LIN {X 0,Y 192.812,Z 326.454,A -85,B 0,C 180,E1 -21972.633,E2 -21972.633} C_VEL
LIN {X 0,Y 192.759,Z 326.462,A -85,B 0,C 180,E1 -21976.959,E2 -21976.959} C_VEL
LIN {X 0,Y 192.618,Z 326.481,A -85,B 0,C 180,E1 -21981.4,E2 -21981.4} C_VEL
LIN {X 0,Y 192.649,Z 326.477,A -85,B 0,C 180,E1 -21984.213,E2 -21984.213} C_VEL
LIN {X 0,Y 192.646,Z 326.478,A -85,B 0,C 180,E1 -21988.889,E2 -21988.889} C_VEL
LIN {X 0,Y 192.627,Z 326.525,A -85,B 0,C 180,E1 -21991.327,E2 -21991.327} C_VEL
LIN {X 0,Y 193.973,Z 330.689,A -85,B 0,C 180,E1 -21995.112,E2 -21995.112} C_VEL
LIN {X 0,Y 197.718,Z 336.194,A -85,B 0,C 180,E1 -21997.257,E2 -21997.257} C_VEL
LIN {X 0,Y 199.002,Z 337.882,A -85,B 0,C 180,E1 -21997.932,E2 -21997.932} C_VEL
LIN {X 0,Y 202.174,Z 342.489,A -85,B 0,C 180,E1 -21999.538,E2 -21999.538} C_VEL
LIN {X 0,Y 207.22,Z 350.444,A -85,B 0,C 180,E1 -22001.911,E2 -22001.911} C_VEL
LIN {X 0,Y 210.777,Z 356.31,A -85,B 0,C 180,E1 -22003.459,E2 -22003.459} C_VEL
LIN {X 0,Y 216.071,Z 365.771,A -85,B 0,C 180,E1 -22005.619,E2 -22005.619} C_VEL
LIN {X 0,Y 220.821,Z 375.163,A -85,B 0,C 180,E1 -22007.434,E2 -22007.434} C_VEL
LIN {X 0,Y 226.552,Z 388.01,A -85,B 0,C 180,E1 -22009.515,E2 -22009.515} C_VEL
LIN {X 0,Y 226.643,Z 388.254,A -85,B 0,C 180,E1 -22009.549,E2 -22009.549} C_VEL
LIN {X 0,Y 227.386,Z 391.769,A -85,B 0,C 180,E1 -22009.885,E2 -22009.885} C_VEL
LIN {X 0,Y 227.296,Z 396.569,A -85,B 0,C 180,E1 -22010.071,E2 -22010.071} C_VEL
LIN {X 0,Y 225.976,Z 403.4,A -85,B 0,C 180,E1 -22010.046,E2 -22010.046} C_VEL
LIN {X 0,Y 222.803,Z 415.633,A -85,B 0,C 180,E1 -22009.796,E2 -22009.796} C_VEL
LIN {X 0,Y 222.248,Z 419.787,A -85,B 0,C 180,E1 -22009.842,E2 -22009.842} C_VEL
LIN {X 0,Y 220.74,Z 442.418,A -85,B 0,C 180,E1 -22010.562,E2 -22010.562} C_VEL
LIN {X 0,Y 218.905,Z 456.037,A -85,B 0,C 180,E1 -22011.297,E2 -22011.297} C_VEL
LIN {X 0,Y 216.473,Z 467.79,A -85,B 0,C 180,E1 -22012.208,E2 -22012.208} C_VEL
LIN {X 0,Y 213.017,Z 480.41,A -85,B 0,C 180,E1 -22013.568,E2 -22013.568} C_VEL
LIN {X 0,Y 209.487,Z 491.624,A -85,B 0,C 180,E1 -22015.227,E2 -22015.227} C_VEL
LIN {X 0,Y 205.624,Z 501.768,A -85,B 0,C 180,E1 -22017.139,E2 -22017.139} C_VEL
LIN {X 0,Y 202.052,Z 510.095,A -85,B 0,C 180,E1 -22019.132,E2 -22019.132} C_VEL
LIN {X 0,Y 197.643,Z 519.156,A -85,B 0,C 180,E1 -22021.89,E2 -22021.89} C_VEL
LIN {X 0,Y 194.46,Z 525.362,A -85,B 0,C 180,E1 -22024.297,E2 -22024.297} C_VEL
LIN {X 0,Y 191.313,Z 531.467,A -85,B 0,C 180,E1 -22027.311,E2 -22027.311} C_VEL
LIN {X 0,Y 188.552,Z 536.333,A -85,B 0,C 180,E1 -22030.399,E2 -22030.399} C_VEL
LIN {X 0,Y 186.292,Z 540.098,A -85,B 0,C 180,E1 -22033.563,E2 -22033.563} C_VEL
LIN {X 0,Y 184.741,Z 542.869,A -85,B 0,C 180,E1 -22036.805,E2 -22036.805} C_VEL
LIN {X 0,Y 183.512,Z 545.134,A -85,B 0,C 180,E1 -22041.188,E2 -22041.188} C_VEL
LIN {X 0,Y 183.214,Z 545.672,A -85,B 0,C 180,E1 -22043.391,E2 -22043.391} C_VEL
LIN {X 0,Y 183.158,Z 545.528,A -85,B 0,C 180,E1 -22047.8,E2 -22047.8} C_VEL
LIN {X 0,Y 183.324,Z 544.879,A -85,B 0,C 180,E1 -22049.999,E2 -22049.999} C_VEL
LIN {X 0,Y 183.155,Z 542.674,A -85,B 0,C 180,E1 -22053.907,E2 -22053.907} C_VEL
LIN {X 0,Y 183.36,Z 539.178,A -85,B 0,C 180,E1 -22057.709,E2 -22057.709} C_VEL
LIN {X 0,Y 183.873,Z 534.991,A -85,B 0,C 180,E1 -22061.017,E2 -22061.017} C_VEL
LIN {X 0,Y 185.089,Z 528.586,A -85,B 0,C 180,E1 -22064.85,E2 -22064.85} C_VEL
LIN {X 0,Y 186.807,Z 521.607,A -85,B 0,C 180,E1 -22068.081,E2 -22068.081} C_VEL
LIN {X 0,Y 188.819,Z 513.433,A -85,B 0,C 180,E1 -22071.069,E2 -22071.069} C_VEL
LIN {X 0,Y 191.033,Z 503.806,A -85,B 0,C 180,E1 -22073.87,E2 -22073.87} C_VEL
LIN {X 0,Y 193.448,Z 493.911,A -85,B 0,C 180,E1 -22076.135,E2 -22076.135} C_VEL
LIN {X 0,Y 195.816,Z 482.985,A -85,B 0,C 180,E1 -22078.103,E2 -22078.103} C_VEL
LIN {X 0,Y 198.082,Z 470.698,A -85,B 0,C 180,E1 -22079.782,E2 -22079.782} C_VEL
LIN {X 0,Y 200.015,Z 457.808,A -85,B 0,C 180,E1 -22081.069,E2 -22081.069} C_VEL
LIN {X 0,Y 201.423,Z 444.674,A -85,B 0,C 180,E1 -22081.935,E2 -22081.935} C_VEL
LIN {X 0,Y 202.283,Z 426.501,A -85,B 0,C 180,E1 -22082.646,E2 -22082.646} C_VEL
LIN {X 0,Y 203.728,Z 391.931,A -85,B 0,C 180,E1 -22083.797,E2 -22083.797} C_VEL
LIN {X 0,Y 201.201,Z 366.378,A -85,B 0,C 180,E1 -22085.24,E2 -22085.24} C_VEL
LIN {X 0,Y 195.007,Z 350.312,A -85,B 0,C 180,E1 -22087.011,E2 -22087.011} C_VEL
LIN {X 0,Y 188.811,Z 336.625,A -85,B 0,C 180,E1 -22088.828,E2 -22088.828} C_VEL
LIN {X 0,Y 186.825,Z 332.463,A -85,B 0,C 180,E1 -22089.479,E2 -22089.479} C_VEL
LIN {X 0,Y 185.486,Z 327.381,A -85,B 0,C 180,E1 -22092.364,E2 -22092.364} C_VEL
LIN {X 0,Y 185.455,Z 327.384,A -85,B 0,C 180,E1 -22096.989,E2 -22096.989} C_VEL
LIN {X 0,Y 185.466,Z 327.383,A -85,B 0,C 180,E1 -22099.894,E2 -22099.894} C_VEL
LIN {X 0,Y 185.504,Z 327.38,A -85,B 0,C 180,E1 -22102.71,E2 -22102.71} C_VEL
LIN {X 0,Y 185.544,Z 327.374,A -85,B 0,C 180,E1 -22107.974,E2 -22107.974} C_VEL
LIN {X 0,Y 185.58,Z 327.371,A -85,B 0,C 180,E1 -22110.575,E2 -22110.575} C_VEL
LIN {X 0,Y 185.586,Z 327.368,A -85,B 0,C 180,E1 -22115.382,E2 -22115.382} C_VEL
LIN {X 0,Y 185.672,Z 327.356,A -85,B 0,C 180,E1 -22121.132,E2 -22121.132} C_VEL
LIN {X 0,Y 185.693,Z 327.354,A -85,B 0,C 180,E1 -22124.637,E2 -22124.637} C_VEL
LIN {X 0,Y 185.921,Z 327.301,A -85,B 0,C 180,E1 -22129.358,E2 -22129.358} C_VEL
LIN {X 0,Y 185.957,Z 327.322,A -85,B 0,C 180,E1 -22133.489,E2 -22133.489} C_VEL
LIN {X 0,Y 186.204,Z 327.27,A -85,B 0,C 180,E1 -22137.836,E2 -22137.836} C_VEL
LIN {X 0,Y 186.401,Z 327.242,A -85,B 0,C 180,E1 -22140,E2 -22140} C_VEL
LIN {X 0,Y 185.911,Z 327.327,A -85,B 0,C 180,E1 -22144.336,E2 -22144.336} C_VEL
LIN {X 0,Y 185.973,Z 327.298,A -85,B 0,C 180,E1 -22148.694,E2 -22148.694} C_VEL
LIN {X 0,Y 185.726,Z 327.345,A -85,B 0,C 180,E1 -22153.123,E2 -22153.123} C_VEL
LIN {X 0,Y 185.686,Z 327.347,A -85,B 0,C 180,E1 -22157.625,E2 -22157.625} C_VEL
LIN {X 0,Y 185.574,Z 327.354,A -85,B 0,C 180,E1 -22162.254,E2 -22162.254} C_VEL
LIN {X 0,Y 185.557,Z 327.366,A -85,B 0,C 180,E1 -22167.032,E2 -22167.032} C_VEL
LIN {X 0,Y 185.576,Z 327.347,A -85,B 0,C 180,E1 -22169.493,E2 -22169.493} C_VEL
LIN {X 0,Y 185.496,Z 327.379,A -85,B 0,C 180,E1 -22174.632,E2 -22174.632} C_VEL
LIN {X 0,Y 185.502,Z 327.365,A -85,B 0,C 180,E1 -22177.313,E2 -22177.313} C_VEL
LIN {X 0,Y 185.466,Z 327.372,A -85,B 0,C 180,E1 -22180.725,E2 -22180.725} C_VEL
LIN {X 0,Y 185.452,Z 327.368,A -85,B 0,C 180,E1 -22186.057,E2 -22186.057} C_VEL
LIN {X 0,Y 185.453,Z 327.382,A -85,B 0,C 180,E1 -22189.893,E2 -22189.893} C_VEL
LIN {X 0,Y 185.498,Z 327.371,A -85,B 0,C 180,E1 -22192.714,E2 -22192.714} C_VEL
LIN {X 0,Y 185.528,Z 327.373,A -85,B 0,C 180,E1 -22197.973,E2 -22197.973} C_VEL
LIN {X 0,Y 185.542,Z 327.365,A -85,B 0,C 180,E1 -22200.598,E2 -22200.598} C_VEL
LIN {X 0,Y 186.69,Z 330.413,A -85,B 0,C 180,E1 -22201.032,E2 -22201.032} C_VEL
LIN {X 0,Y 188.069,Z 332.496,A -85,B 0,C 180,E1 -22201.42,E2 -22201.42} C_VEL
LIN {X 0,Y 196.411,Z 347.504,A -85,B 0,C 180,E1 -22203.72,E2 -22203.72} C_VEL
LIN {X 0,Y 202.022,Z 359.493,A -85,B 0,C 180,E1 -22205.209,E2 -22205.209} C_VEL
LIN {X 0,Y 204.649,Z 366.895,A -85,B 0,C 180,E1 -22205.944,E2 -22205.944} C_VEL
LIN {X 0,Y 202.081,Z 428.474,A -85,B 0,C 180,E1 -22208.047,E2 -22208.047} C_VEL
LIN {X 0,Y 201.051,Z 441.583,A -85,B 0,C 180,E1 -22208.871,E2 -22208.871} C_VEL
LIN {X 0,Y 199.598,Z 454.209,A -85,B 0,C 180,E1 -22210.057,E2 -22210.057} C_VEL
LIN {X 0,Y 197.638,Z 466.289,A -85,B 0,C 180,E1 -22211.604,E2 -22211.604} C_VEL
LIN {X 0,Y 195.28,Z 476.551,A -85,B 0,C 180,E1 -22213.268,E2 -22213.268} C_VEL
LIN {X 0,Y 193.014,Z 487.091,A -85,B 0,C 180,E1 -22215.504,E2 -22215.504} C_VEL
LIN {X 0,Y 190.864,Z 495.73,A -85,B 0,C 180,E1 -22217.777,E2 -22217.777} C_VEL
LIN {X 0,Y 188.847,Z 503.679,A -85,B 0,C 180,E1 -22220.36,E2 -22220.36} C_VEL
LIN {X 0,Y 186.807,Z 511.476,A -85,B 0,C 180,E1 -22223.52,E2 -22223.52} C_VEL
LIN {X 0,Y 185.331,Z 517.701,A -85,B 0,C 180,E1 -22226.74,E2 -22226.74} C_VEL
LIN {X 0,Y 184.203,Z 522.666,A -85,B 0,C 180,E1 -22230.001,E2 -22230.001} C_VEL
LIN {X 0,Y 183.672,Z 526.498,A -85,B 0,C 180,E1 -22233.291,E2 -22233.291} C_VEL
LIN {X 0,Y 183.237,Z 529.33,A -85,B 0,C 180,E1 -22236.608,E2 -22236.608} C_VEL
LIN {X 0,Y 183.023,Z 531.63,A -85,B 0,C 180,E1 -22241.07,E2 -22241.07} C_VEL
LIN {X 0,Y 183.204,Z 532.178,A -85,B 0,C 180,E1 -22243.308,E2 -22243.308} C_VEL
LIN {X 0,Y 183.963,Z 532.117,A -85,B 0,C 180,E1 -22247.239,E2 -22247.239} C_VEL
LIN {X 0,Y 184.736,Z 531.333,A -85,B 0,C 180,E1 -22250.023,E2 -22250.023} C_VEL
LIN {X 0,Y 185.631,Z 530.231,A -85,B 0,C 180,E1 -22252.248,E2 -22252.248} C_VEL
LIN {X 0,Y 187.811,Z 527.22,A -85,B 0,C 180,E1 -22256.092,E2 -22256.092} C_VEL
LIN {X 0,Y 190.685,Z 522.809,A -85,B 0,C 180,E1 -22259.84,E2 -22259.84} C_VEL
LIN {X 0,Y 193.663,Z 517.741,A -85,B 0,C 180,E1 -22262.981,E2 -22262.981} C_VEL
LIN {X 0,Y 197.251,Z 511.31,A -85,B 0,C 180,E1 -22266.008,E2 -22266.008} C_VEL
LIN {X 0,Y 201.297,Z 503.198,A -85,B 0,C 180,E1 -22268.936,E2 -22268.936} C_VEL
LIN {X 0,Y 205.47,Z 494.072,A -85,B 0,C 180,E1 -22271.474,E2 -22271.474} C_VEL
LIN {X 0,Y 209.165,Z 484.669,A -85,B 0,C 180,E1 -22273.536,E2 -22273.536} C_VEL
LIN {X 0,Y 212.535,Z 474.439,A -85,B 0,C 180,E1 -22275.313,E2 -22275.313} C_VEL
LIN {X 0,Y 215.81,Z 462.836,A -85,B 0,C 180,E1 -22276.853,E2 -22276.853} C_VEL
LIN {X 0,Y 218.392,Z 450.783,A -85,B 0,C 180,E1 -22278.084,E2 -22278.084} C_VEL
LIN {X 0,Y 220.382,Z 437.633,A -85,B 0,C 180,E1 -22279.034,E2 -22279.034} C_VEL
LIN {X 0,Y 221.649,Z 425.884,A -85,B 0,C 180,E1 -22279.552,E2 -22279.552} C_VEL
LIN {X 0,Y 224.092,Z 386.328,A -85,B 0,C 180,E1 -22280.719,E2 -22280.719} C_VEL
LIN {X 0,Y 218.281,Z 374.069,A -85,B 0,C 180,E1 -22282.866,E2 -22282.866} C_VEL
LIN {X 0,Y 213.163,Z 365.33,A -85,B 0,C 180,E1 -22284.835,E2 -22284.835} C_VEL
LIN {X 0,Y 206.43,Z 355.119,A -85,B 0,C 180,E1 -22287.646,E2 -22287.646} C_VEL
LIN {X 0,Y 203.304,Z 350.827,A -85,B 0,C 180,E1 -22289.056,E2 -22289.056} C_VEL
LIN {X 0,Y 200.397,Z 346.848,A -85,B 0,C 180,E1 -22290.451,E2 -22290.451} C_VEL
LIN {X 0,Y 197.599,Z 343.03,A -85,B 0,C 180,E1 -22291.884,E2 -22291.884} C_VEL
LIN {X 0,Y 194.884,Z 339.672,A -85,B 0,C 180,E1 -22293.351,E2 -22293.351} C_VEL
LIN {X 0,Y 194.108,Z 338.344,A -85,B 0,C 180,E1 -22293.816,E2 -22293.816} C_VEL
LIN {X 0,Y 191.552,Z 336.002,A -85,B 0,C 180,E1 -22295.269,E2 -22295.269} C_VEL
LIN {X 0,Y 189.931,Z 332.999,A -85,B 0,C 180,E1 -22296.363,E2 -22296.363} C_VEL
LIN {X 0,Y 187.274,Z 331.168,A -85,B 0,C 180,E1 -22298.031,E2 -22298.031} C_VEL
LIN {X 0,Y 185.951,Z 328.94,A -85,B 0,C 180,E1 -22299.031,E2 -22299.031} C_VEL
LIN {X 0,Y 185.571,Z 327.359,A -85,B 0,C 180,E1 -22299.494,E2 -22299.494} C_VEL
LIN {X 0,Y 185.691,Z 327.352,A -85,B 0,C 180,E1 -22302.376,E2 -22302.376} C_VEL
LIN {X 0,Y 185.767,Z 327.346,A -85,B 0,C 180,E1 -22306.88,E2 -22306.88} C_VEL
LIN {X 0,Y 186.031,Z 327.313,A -85,B 0,C 180,E1 -22311.309,E2 -22311.309} C_VEL
LIN {X 0,Y 186.209,Z 327.275,A -85,B 0,C 180,E1 -22317.837,E2 -22317.837} C_VEL
LIN {X 0,Y 186.406,Z 327.262,A -85,B 0,C 180,E1 -22320,E2 -22320} C_VEL
LIN {X 0,Y 185.926,Z 327.319,A -85,B 0,C 180,E1 -22324.336,E2 -22324.336} C_VEL
LIN {X 0,Y 186.011,Z 327.306,A -85,B 0,C 180,E1 -22328.693,E2 -22328.693} C_VEL
LIN {X 0,Y 185.736,Z 327.34,A -85,B 0,C 180,E1 -22333.123,E2 -22333.123} C_VEL
LIN {X 0,Y 185.692,Z 327.347,A -85,B 0,C 180,E1 -22337.625,E2 -22337.625} C_VEL
LIN {X 0,Y 185.58,Z 327.366,A -85,B 0,C 180,E1 -22342.254,E2 -22342.254} C_VEL
LIN {X 0,Y 185.561,Z 327.369,A -85,B 0,C 180,E1 -22347.033,E2 -22347.033} C_VEL
LIN {X 0,Y 185.635,Z 327.541,A -85,B 0,C 180,E1 -22348.245,E2 -22348.245} C_VEL
LIN {X 0,Y 186.616,Z 330.253,A -85,B 0,C 180,E1 -22351.029,E2 -22351.029} C_VEL
LIN {X 0,Y 189.543,Z 334.692,A -85,B 0,C 180,E1 -22353.09,E2 -22353.09} C_VEL
LIN {X 0,Y 191.645,Z 337.156,A -85,B 0,C 180,E1 -22354.401,E2 -22354.401} C_VEL
LIN {X 0,Y 195.551,Z 342.71,A -85,B 0,C 180,E1 -22356.706,E2 -22356.706} C_VEL
LIN {X 0,Y 200.091,Z 349.688,A -85,B 0,C 180,E1 -22359.135,E2 -22359.135} C_VEL
LIN {X 0,Y 204.237,Z 356.412,A -85,B 0,C 180,E1 -22361.159,E2 -22361.159} C_VEL
LIN {X 0,Y 208.864,Z 364.216,A -85,B 0,C 180,E1 -22363.239,E2 -22363.239} C_VEL
LIN {X 0,Y 214.944,Z 375.86,A -85,B 0,C 180,E1 -22365.78,E2 -22365.78} C_VEL
LIN {X 0,Y 221.35,Z 390.268,A -85,B 0,C 180,E1 -22368.276,E2 -22368.276} C_VEL
LIN {X 0,Y 222.965,Z 394.781,A -85,B 0,C 180,E1 -22368.906,E2 -22368.906} C_VEL
LIN {X 0,Y 223.453,Z 400.102,A -85,B 0,C 180,E1 -22369.269,E2 -22369.269} C_VEL
LIN {X 0,Y 222.248,Z 419.787,A -85,B 0,C 180,E1 -22369.842,E2 -22369.842} C_VEL
LIN {X 0,Y 221.384,Z 425.64,A -85,B 0,C 180,E1 -22369.875,E2 -22369.875} C_VEL
LIN {X 0,Y 215.811,Z 444.62,A -85,B 0,C 180,E1 -22369.47,E2 -22369.47} C_VEL
LIN {X 0,Y 214.644,Z 450.37,A -85,B 0,C 180,E1 -22369.66,E2 -22369.66} C_VEL
LIN {X 0,Y 212.192,Z 463.375,A -85,B 0,C 180,E1 -22370.55,E2 -22370.55} C_VEL
LIN {X 0,Y 208.901,Z 476.223,A -85,B 0,C 180,E1 -22371.816,E2 -22371.816} C_VEL
LIN {X 0,Y 205.574,Z 486.943,A -85,B 0,C 180,E1 -22373.253,E2 -22373.253} C_VEL
LIN {X 0,Y 201.41,Z 497.92,A -85,B 0,C 180,E1 -22375.152,E2 -22375.152} C_VEL
LIN {X 0,Y 196.79,Z 508.622,A -85,B 0,C 180,E1 -22377.608,E2 -22377.608} C_VEL
LIN {X 0,Y 192.878,Z 516.543,A -85,B 0,C 180,E1 -22379.932,E2 -22379.932} C_VEL
LIN {X 0,Y 188.701,Z 524.322,A -85,B 0,C 180,E1 -22382.855,E2 -22382.855} C_VEL
LIN {X 0,Y 184.775,Z 531.477,A -85,B 0,C 180,E1 -22386.46,E2 -22386.46} C_VEL
LIN {X 0,Y 181.842,Z 536.282,A -85,B 0,C 180,E1 -22389.644,E2 -22389.644} C_VEL
LIN {X 0,Y 179.473,Z 539.992,A -85,B 0,C 180,E1 -22392.92,E2 -22392.92} C_VEL
LIN {X 0,Y 177.801,Z 542.712,A -85,B 0,C 180,E1 -22396.28,E2 -22396.28} C_VEL
LIN {X 0,Y 176.474,Z 544.927,A -85,B 0,C 180,E1 -22400.833,E2 -22400.833} C_VEL
LIN {X 0,Y 176.142,Z 545.418,A -85,B 0,C 180,E1 -22403.125,E2 -22403.125} C_VEL
LIN {X 0,Y 176.054,Z 545.227,A -85,B 0,C 180,E1 -22407.711,E2 -22407.711} C_VEL
LIN {X 0,Y 176.243,Z 544.555,A -85,B 0,C 180,E1 -22409.999,E2 -22409.999} C_VEL
LIN {X 0,Y 176.07,Z 542.538,A -85,B 0,C 180,E1 -22413.704,E2 -22413.704} C_VEL
LIN {X 0,Y 176.316,Z 538.726,A -85,B 0,C 180,E1 -22418.019,E2 -22418.019} C_VEL
LIN {X 0,Y 176.881,Z 534.483,A -85,B 0,C 180,E1 -22421.458,E2 -22421.458} C_VEL
LIN {X 0,Y 178.182,Z 528.015,A -85,B 0,C 180,E1 -22425.44,E2 -22425.44} C_VEL
LIN {X 0,Y 179.981,Z 520.946,A -85,B 0,C 180,E1 -22428.792,E2 -22428.792} C_VEL
LIN {X 0,Y 181.807,Z 514.255,A -85,B 0,C 180,E1 -22431.344,E2 -22431.344} C_VEL
LIN {X 0,Y 184.017,Z 504.925,A -85,B 0,C 180,E1 -22434.239,E2 -22434.239} C_VEL
LIN {X 0,Y 186.763,Z 494.121,A -85,B 0,C 180,E1 -22436.843,E2 -22436.843} C_VEL
LIN {X 0,Y 189.215,Z 483.345,A -85,B 0,C 180,E1 -22438.871,E2 -22438.871} C_VEL
LIN {X 0,Y 191.571,Z 471.237,A -85,B 0,C 180,E1 -22440.597,E2 -22440.597} C_VEL
LIN {X 0,Y 193.57,Z 458.603,A -85,B 0,C 180,E1 -22441.918,E2 -22441.918} C_VEL
LIN {X 0,Y 195.02,Z 446.072,A -85,B 0,C 180,E1 -22442.818,E2 -22442.818} C_VEL
LIN {X 0,Y 195.868,Z 430.553,A -85,B 0,C 180,E1 -22443.486,E2 -22443.486} C_VEL
LIN {X 0,Y 197.525,Z 391.561,A -85,B 0,C 180,E1 -22444.825,E2 -22444.825} C_VEL
LIN {X 0,Y 195.125,Z 368.319,A -85,B 0,C 180,E1 -22446.22,E2 -22446.22} C_VEL
LIN {X 0,Y 189.403,Z 353.427,A -85,B 0,C 180,E1 -22447.953,E2 -22447.953} C_VEL
LIN {X 0,Y 183.653,Z 340.606,A -85,B 0,C 180,E1 -22449.74,E2 -22449.74} C_VEL
LIN {X 0,Y 180.545,Z 334.628,A -85,B 0,C 180,E1 -22450.724,E2 -22450.724} C_VEL
LIN {X 0,Y 179.412,Z 332.121,A -85,B 0,C 180,E1 -22451.162,E2 -22451.162} C_VEL
LIN {X 0,Y 178.406,Z 328.263,A -85,B 0,C 180,E1 -22453.563,E2 -22453.563} C_VEL
LIN {X 0,Y 178.401,Z 328.267,A -85,B 0,C 180,E1 -22458.458,E2 -22458.458} C_VEL
LIN {X 0,Y 178.421,Z 328.264,A -85,B 0,C 180,E1 -22463.782,E2 -22463.782} C_VEL
LIN {X 0,Y 178.485,Z 328.256,A -85,B 0,C 180,E1 -22466.546,E2 -22466.546} C_VEL
LIN {X 0,Y 178.521,Z 328.25,A -85,B 0,C 180,E1 -22470.005,E2 -22470.005} C_VEL
LIN {X 0,Y 178.533,Z 328.246,A -85,B 0,C 180,E1 -22474.875,E2 -22474.875} C_VEL
LIN {X 0,Y 178.621,Z 328.236,A -85,B 0,C 180,E1 -22480.783,E2 -22480.783} C_VEL
LIN {X 0,Y 178.658,Z 328.221,A -85,B 0,C 180,E1 -22486.347,E2 -22486.347} C_VEL
LIN {X 0,Y 178.956,Z 328.181,A -85,B 0,C 180,E1 -22490.962,E2 -22490.962} C_VEL
LIN {X 0,Y 179.15,Z 328.148,A -85,B 0,C 180,E1 -22497.751,E2 -22497.751} C_VEL
LIN {X 0,Y 179.364,Z 328.117,A -85,B 0,C 180,E1 -22500,E2 -22500} C_VEL
LIN {X 0,Y 178.858,Z 328.205,A -85,B 0,C 180,E1 -22504.507,E2 -22504.507} C_VEL
LIN {X 0,Y 178.903,Z 328.175,A -85,B 0,C 180,E1 -22509.04,E2 -22509.04} C_VEL
LIN {X 0,Y 178.654,Z 328.227,A -85,B 0,C 180,E1 -22513.652,E2 -22513.652} C_VEL
LIN {X 0,Y 178.617,Z 328.214,A -85,B 0,C 180,E1 -22519.214,E2 -22519.214} C_VEL
LIN {X 0,Y 178.516,Z 328.248,A -85,B 0,C 180,E1 -22525.114,E2 -22525.114} C_VEL
LIN {X 0,Y 178.52,Z 328.223,A -85,B 0,C 180,E1 -22529.994,E2 -22529.994} C_VEL
LIN {X 0,Y 178.482,Z 328.25,A -85,B 0,C 180,E1 -22534.22,E2 -22534.22} C_VEL
LIN {X 0,Y 178.391,Z 328.243,A -85,B 0,C 180,E1 -22539.075,E2 -22539.075} C_VEL
LIN {X 0,Y 178.394,Z 328.26,A -85,B 0,C 180,E1 -22542.046,E2 -22542.046} C_VEL
LIN {X 0,Y 178.388,Z 328.249,A -85,B 0,C 180,E1 -22545.165,E2 -22545.165} C_VEL
LIN {X 0,Y 178.394,Z 328.261,A -85,B 0,C 180,E1 -22548.462,E2 -22548.462} C_VEL
LIN {X 0,Y 178.416,Z 328.261,A -85,B 0,C 180,E1 -22553.783,E2 -22553.783} C_VEL
LIN {X 0,Y 178.463,Z 328.253,A -85,B 0,C 180,E1 -22558.549,E2 -22558.549} C_VEL
LIN {X 0,Y 178.486,Z 328.413,A -85,B 0,C 180,E1 -22559.078,E2 -22559.078} C_VEL
LIN {X 0,Y 179.518,Z 331.187,A -85,B 0,C 180,E1 -22559.46,E2 -22559.46} C_VEL
LIN {X 0,Y 181.038,Z 333.344,A -85,B 0,C 180,E1 -22559.918,E2 -22559.918} C_VEL
LIN {X 0,Y 188.944,Z 347.167,A -85,B 0,C 180,E1 -22562.265,E2 -22562.265} C_VEL
LIN {X 0,Y 195.661,Z 360.844,A -85,B 0,C 180,E1 -22564.151,E2 -22564.151} C_VEL
LIN {X 0,Y 198.582,Z 369.012,A -85,B 0,C 180,E1 -22565.012,E2 -22565.012} C_VEL
LIN {X 0,Y 195.826,Z 429.016,A -85,B 0,C 180,E1 -22567.098,E2 -22567.098} C_VEL
LIN {X 0,Y 194.675,Z 442.788,A -85,B 0,C 180,E1 -22568.005,E2 -22568.005} C_VEL
LIN {X 0,Y 193.13,Z 455.173,A -85,B 0,C 180,E1 -22569.22,E2 -22569.22} C_VEL
LIN {X 0,Y 191.258,Z 466.259,A -85,B 0,C 180,E1 -22570.689,E2 -22570.689} C_VEL
LIN {X 0,Y 188.816,Z 476.575,A -85,B 0,C 180,E1 -22572.398,E2 -22572.398} C_VEL
LIN {X 0,Y 186.426,Z 487.157,A -85,B 0,C 180,E1 -22574.7,E2 -22574.7} C_VEL
LIN {X 0,Y 183.967,Z 496.715,A -85,B 0,C 180,E1 -22577.312,E2 -22577.312} C_VEL
LIN {X 0,Y 181.858,Z 504.545,A -85,B 0,C 180,E1 -22579.986,E2 -22579.986} C_VEL
LIN {X 0,Y 179.764,Z 512.194,A -85,B 0,C 180,E1 -22583.265,E2 -22583.265} C_VEL
LIN {X 0,Y 178.248,Z 518.333,A -85,B 0,C 180,E1 -22586.61,E2 -22586.61} C_VEL
LIN {X 0,Y 177.095,Z 523.22,A -85,B 0,C 180,E1 -22590.001,E2 -22590.001} C_VEL
LIN {X 0,Y 176.57,Z 526.98,A -85,B 0,C 180,E1 -22593.424,E2 -22593.424} C_VEL
LIN {X 0,Y 176.105,Z 529.746,A -85,B 0,C 180,E1 -22596.877,E2 -22596.877} C_VEL
LIN {X 0,Y 175.923,Z 531.061,A -85,B 0,C 180,E1 -22599.196,E2 -22599.196} C_VEL
LIN {X 0,Y 175.941,Z 531.981,A -85,B 0,C 180,E1 -22601.522,E2 -22601.522} C_VEL
LIN {X 0,Y 176.172,Z 532.465,A -85,B 0,C 180,E1 -22603.849,E2 -22603.849} C_VEL
LIN {X 0,Y 176.929,Z 532.409,A -85,B 0,C 180,E1 -22607.575,E2 -22607.575} C_VEL
LIN {X 0,Y 177.9,Z 531.517,A -85,B 0,C 180,E1 -22610.828,E2 -22610.828} C_VEL
LIN {X 0,Y 178.894,Z 530.351,A -85,B 0,C 180,E1 -22613.133,E2 -22613.133} C_VEL
LIN {X 0,Y 181.06,Z 527.583,A -85,B 0,C 180,E1 -22616.778,E2 -22616.778} C_VEL
LIN {X 0,Y 184.368,Z 522.785,A -85,B 0,C 180,E1 -22620.972,E2 -22620.972} C_VEL
LIN {X 0,Y 188.19,Z 516.555,A -85,B 0,C 180,E1 -22624.756,E2 -22624.756} C_VEL
LIN {X 0,Y 192.051,Z 509.823,A -85,B 0,C 180,E1 -22627.804,E2 -22627.804} C_VEL
LIN {X 0,Y 196.386,Z 501.542,A -85,B 0,C 180,E1 -22630.687,E2 -22630.687} C_VEL
LIN {X 0,Y 200.529,Z 492.509,A -85,B 0,C 180,E1 -22633.112,E2 -22633.112} C_VEL
LIN {X 0,Y 204.369,Z 482.778,A -85,B 0,C 180,E1 -22635.176,E2 -22635.176} C_VEL
LIN {X 0,Y 207.96,Z 472.084,A -85,B 0,C 180,E1 -22636.955,E2 -22636.955} C_VEL
LIN {X 0,Y 211.264,Z 460.038,A -85,B 0,C 180,E1 -22638.481,E2 -22638.481} C_VEL
LIN {X 0,Y 213.751,Z 448.236,A -85,B 0,C 180,E1 -22639.592,E2 -22639.592} C_VEL
LIN {X 0,Y 215.627,Z 435.138,A -85,B 0,C 180,E1 -22640.486,E2 -22640.486} C_VEL
LIN {X 0,Y 216.929,Z 422.502,A -85,B 0,C 180,E1 -22640.954,E2 -22640.954} C_VEL
LIN {X 0,Y 219.055,Z 388.94,A -85,B 0,C 180,E1 -22641.943,E2 -22641.943} C_VEL
LIN {X 0,Y 213.27,Z 376.764,A -85,B 0,C 180,E1 -22644.221,E2 -22644.221} C_VEL
LIN {X 0,Y 206.554,Z 365.622,A -85,B 0,C 180,E1 -22647.017,E2 -22647.017} C_VEL
LIN {X 0,Y 200.616,Z 356.921,A -85,B 0,C 180,E1 -22649.745,E2 -22649.745} C_VEL
LIN {X 0,Y 197.256,Z 352.324,A -85,B 0,C 180,E1 -22651.432,E2 -22651.432} C_VEL
LIN {X 0,Y 194.692,Z 348.815,A -85,B 0,C 180,E1 -22652.815,E2 -22652.815} C_VEL
LIN {X 0,Y 191.985,Z 345.144,A -85,B 0,C 180,E1 -22654.379,E2 -22654.379} C_VEL
LIN {X 0,Y 188.631,Z 341.293,A -85,B 0,C 180,E1 -22656.436,E2 -22656.436} C_VEL
LIN {X 0,Y 187.551,Z 339.461,A -85,B 0,C 180,E1 -22657.191,E2 -22657.191} C_VEL
LIN {X 0,Y 184.902,Z 337.157,A -85,B 0,C 180,E1 -22658.979,E2 -22658.979} C_VEL
LIN {X 0,Y 183.244,Z 334.042,A -85,B 0,C 180,E1 -22660.342,E2 -22660.342} C_VEL
LIN {X 0,Y 180.561,Z 332.251,A -85,B 0,C 180,E1 -22662.443,E2 -22662.443} C_VEL
LIN {X 0,Y 179.044,Z 329.903,A -85,B 0,C 180,E1 -22663.906,E2 -22663.906} C_VEL
LIN {X 0,Y 178.648,Z 328.22,A -85,B 0,C 180,E1 -22664.455,E2 -22664.455} C_VEL
LIN {X 0,Y 178.897,Z 328.188,A -85,B 0,C 180,E1 -22669.154,E2 -22669.154} C_VEL
LIN {X 0,Y 178.935,Z 328.183,A -85,B 0,C 180,E1 -22673.234,E2 -22673.234} C_VEL
LIN {X 0,Y 179.155,Z 328.154,A -85,B 0,C 180,E1 -22677.752,E2 -22677.752} C_VEL
LIN {X 0,Y 179.37,Z 328.139,A -85,B 0,C 180,E1 -22680,E2 -22680} C_VEL
LIN {X 0,Y 178.875,Z 328.199,A -85,B 0,C 180,E1 -22684.507,E2 -22684.507} C_VEL
LIN {X 0,Y 178.962,Z 328.187,A -85,B 0,C 180,E1 -22689.038,E2 -22689.038} C_VEL
LIN {X 0,Y 178.663,Z 328.226,A -85,B 0,C 180,E1 -22693.652,E2 -22693.652} C_VEL
LIN {X 0,Y 178.623,Z 328.226,A -85,B 0,C 180,E1 -22699.214,E2 -22699.214} C_VEL
LIN {X 0,Y 178.547,Z 328.389,A -85,B 0,C 180,E1 -22704.218,E2 -22704.218} C_VEL
LIN {X 0,Y 178.79,Z 329.503,A -85,B 0,C 180,E1 -22705.374,E2 -22705.374} C_VEL
LIN {X 0,Y 179.919,Z 331.705,A -85,B 0,C 180,E1 -22706.537,E2 -22706.537} C_VEL
LIN {X 0,Y 182.072,Z 333.998,A -85,B 0,C 180,E1 -22708.377,E2 -22708.377} C_VEL
LIN {X 0,Y 184.724,Z 337.012,A -85,B 0,C 180,E1 -22710.431,E2 -22710.431} C_VEL
LIN {X 0,Y 187.504,Z 341.164,A -85,B 0,C 180,E1 -22712.455,E2 -22712.455} C_VEL
LIN {X 0,Y 189.341,Z 343.472,A -85,B 0,C 180,E1 -22713.657,E2 -22713.657} C_VEL
LIN {X 0,Y 193.636,Z 349.968,A -85,B 0,C 180,E1 -22716.304,E2 -22716.304} C_VEL
LIN {X 0,Y 197.297,Z 355.702,A -85,B 0,C 180,E1 -22718.339,E2 -22718.339} C_VEL
LIN {X 0,Y 200.988,Z 361.812,A -85,B 0,C 180,E1 -22720.233,E2 -22720.233} C_VEL
LIN {X 0,Y 205.088,Z 368.897,A -85,B 0,C 180,E1 -22722.181,E2 -22722.181} C_VEL
LIN {X 0,Y 211.007,Z 380.548,A -85,B 0,C 180,E1 -22724.802,E2 -22724.802} C_VEL
LIN {X 0,Y 216.816,Z 393.894,A -85,B 0,C 180,E1 -22727.202,E2 -22727.202} C_VEL
LIN {X 0,Y 218.117,Z 397.454,A -85,B 0,C 180,E1 -22727.734,E2 -22727.734} C_VEL
LIN {X 0,Y 218.387,Z 401.64,A -85,B 0,C 180,E1 -22728.004,E2 -22728.004} C_VEL
LIN {X 0,Y 215.767,Z 441.266,A -85,B 0,C 180,E1 -22729.217,E2 -22729.217} C_VEL
LIN {X 0,Y 214.644,Z 450.37,A -85,B 0,C 180,E1 -22729.66,E2 -22729.66} C_VEL
LIN {X 0,Y 213.27,Z 456.065,A -85,B 0,C 180,E1 -22729.876,E2 -22729.876} C_VEL
LIN {X 0,Y 209.323,Z 465.152,A -85,B 0,C 180,E1 -22730.035,E2 -22730.035} C_VEL
LIN {X 0,Y 204.86,Z 473.938,A -85,B 0,C 180,E1 -22730.359,E2 -22730.359} C_VEL
LIN {X 0,Y 202.69,Z 479.163,A -85,B 0,C 180,E1 -22730.844,E2 -22730.844} C_VEL
LIN {X 0,Y 198.523,Z 491.391,A -85,B 0,C 180,E1 -22732.681,E2 -22732.681} C_VEL
LIN {X 0,Y 194.292,Z 501.467,A -85,B 0,C 180,E1 -22734.636,E2 -22734.636} C_VEL
LIN {X 0,Y 190.009,Z 510.567,A -85,B 0,C 180,E1 -22736.936,E2 -22736.936} C_VEL
LIN {X 0,Y 185.253,Z 519.458,A -85,B 0,C 180,E1 -22739.823,E2 -22739.823} C_VEL
LIN {X 0,Y 181.06,Z 526.74,A -85,B 0,C 180,E1 -22742.927,E2 -22742.927} C_VEL
LIN {X 0,Y 177.177,Z 533.196,A -85,B 0,C 180,E1 -22746.629,E2 -22746.629} C_VEL
LIN {X 0,Y 174.304,Z 537.567,A -85,B 0,C 180,E1 -22749.956,E2 -22749.956} C_VEL
LIN {X 0,Y 171.955,Z 540.887,A -85,B 0,C 180,E1 -22753.375,E2 -22753.375} C_VEL
LIN {X 0,Y 170.057,Z 543.833,A -85,B 0,C 180,E1 -22758.074,E2 -22758.074} C_VEL
LIN {X 0,Y 169.456,Z 544.712,A -85,B 0,C 180,E1 -22760.45,E2 -22760.45} C_VEL
LIN {X 0,Y 168.932,Z 545.236,A -85,B 0,C 180,E1 -22765.226,E2 -22765.226} C_VEL
LIN {X 0,Y 168.952,Z 544.925,A -85,B 0,C 180,E1 -22767.615,E2 -22767.615} C_VEL
LIN {X 0,Y 169.144,Z 544.228,A -85,B 0,C 180,E1 -22769.999,E2 -22769.999} C_VEL
LIN {X 0,Y 168.976,Z 542.428,A -85,B 0,C 180,E1 -22773.427,E2 -22773.427} C_VEL
LIN {X 0,Y 169.15,Z 539.47,A -85,B 0,C 180,E1 -22777.159,E2 -22777.159} C_VEL
LIN {X 0,Y 169.63,Z 535.544,A -85,B 0,C 180,E1 -22780.744,E2 -22780.744} C_VEL
LIN {X 0,Y 170.559,Z 530.459,A -85,B 0,C 180,E1 -22784.313,E2 -22784.313} C_VEL
LIN {X 0,Y 172.259,Z 524.069,A -85,B 0,C 180,E1 -22787.817,E2 -22787.817} C_VEL
LIN {X 0,Y 174.075,Z 517.531,A -85,B 0,C 180,E1 -22790.686,E2 -22790.686} C_VEL
LIN {X 0,Y 176.124,Z 509.635,A -85,B 0,C 180,E1 -22793.517,E2 -22793.517} C_VEL
LIN {X 0,Y 178.676,Z 499.984,A -85,B 0,C 180,E1 -22796.263,E2 -22796.263} C_VEL
LIN {X 0,Y 181.346,Z 489.273,A -85,B 0,C 180,E1 -22798.657,E2 -22798.657} C_VEL
LIN {X 0,Y 183.701,Z 478.932,A -85,B 0,C 180,E1 -22800.457,E2 -22800.457} C_VEL
LIN {X 0,Y 185.881,Z 467.736,A -85,B 0,C 180,E1 -22801.959,E2 -22801.959} C_VEL
LIN {X 0,Y 187.748,Z 455.138,A -85,B 0,C 180,E1 -22803.192,E2 -22803.192} C_VEL
LIN {X 0,Y 189.097,Z 442.028,A -85,B 0,C 180,E1 -22804.05,E2 -22804.05} C_VEL
LIN {X 0,Y 191.417,Z 392.633,A -85,B 0,C 180,E1 -22805.848,E2 -22805.848} C_VEL
LIN {X 0,Y 189.205,Z 370.499,A -85,B 0,C 180,E1 -22807.232,E2 -22807.232} C_VEL
LIN {X 0,Y 183.098,Z 354.582,A -85,B 0,C 180,E1 -22809.206,E2 -22809.206} C_VEL
LIN {X 0,Y 178.04,Z 343.54,A -85,B 0,C 180,E1 -22810.874,E2 -22810.874} C_VEL
LIN {X 0,Y 173.759,Z 335.362,A -85,B 0,C 180,E1 -22812.332,E2 -22812.332} C_VEL
LIN {X 0,Y 172.051,Z 331.735,A -85,B 0,C 180,E1 -22813.043,E2 -22813.043} C_VEL
LIN {X 0,Y 171.375,Z 329.137,A -85,B 0,C 180,E1 -22814.814,E2 -22814.814} C_VEL
LIN {X 0,Y 171.333,Z 329.145,A -85,B 0,C 180,E1 -22818.98,E2 -22818.98} C_VEL
LIN {X 0,Y 171.385,Z 329.139,A -85,B 0,C 180,E1 -22822.04,E2 -22822.04} C_VEL
LIN {X 0,Y 171.397,Z 329.137,A -85,B 0,C 180,E1 -22825.091,E2 -22825.091} C_VEL
LIN {X 0,Y 171.447,Z 329.132,A -85,B 0,C 180,E1 -22830.533,E2 -22830.533} C_VEL
LIN {X 0,Y 171.456,Z 329.129,A -85,B 0,C 180,E1 -22835.801,E2 -22835.801} C_VEL
LIN {X 0,Y 171.577,Z 329.113,A -85,B 0,C 180,E1 -22840.871,E2 -22840.871} C_VEL
LIN {X 0,Y 171.576,Z 329.106,A -85,B 0,C 180,E1 -22845.772,E2 -22845.772} C_VEL
LIN {X 0,Y 171.885,Z 329.056,A -85,B 0,C 180,E1 -22850.586,E2 -22850.586} C_VEL
LIN {X 0,Y 171.817,Z 329.08,A -85,B 0,C 180,E1 -22855.307,E2 -22855.307} C_VEL
LIN {X 0,Y 172.327,Z 328.992,A -85,B 0,C 180,E1 -22859.999,E2 -22859.999} C_VEL
LIN {X 0,Y 171.806,Z 329.083,A -85,B 0,C 180,E1 -22864.692,E2 -22864.692} C_VEL
LIN {X 0,Y 171.841,Z 329.052,A -85,B 0,C 180,E1 -22869.415,E2 -22869.415} C_VEL
LIN {X 0,Y 171.572,Z 329.112,A -85,B 0,C 180,E1 -22874.227,E2 -22874.227} C_VEL
LIN {X 0,Y 171.536,Z 329.092,A -85,B 0,C 180,E1 -22879.557,E2 -22879.557} C_VEL
LIN {X 0,Y 171.455,Z 329.127,A -85,B 0,C 180,E1 -22885.609,E2 -22885.609} C_VEL
LIN {X 0,Y 171.438,Z 329.105,A -85,B 0,C 180,E1 -22890.587,E2 -22890.587} C_VEL
LIN {X 0,Y 171.389,Z 329.134,A -85,B 0,C 180,E1 -22895.035,E2 -22895.035} C_VEL
LIN {X 0,Y 171.353,Z 329.118,A -85,B 0,C 180,E1 -22898.807,E2 -22898.807} C_VEL
LIN {X 0,Y 171.316,Z 329.136,A -85,B 0,C 180,E1 -22904.218,E2 -22904.218} C_VEL
LIN {X 0,Y 171.327,Z 329.144,A -85,B 0,C 180,E1 -22908.98,E2 -22908.98} C_VEL
LIN {X 0,Y 171.357,Z 329.129,A -85,B 0,C 180,E1 -22912.035,E2 -22912.035} C_VEL
LIN {X 0,Y 171.444,Z 329.127,A -85,B 0,C 180,E1 -22917.298,E2 -22917.298} C_VEL
LIN {X 0,Y 172.418,Z 331.942,A -85,B 0,C 180,E1 -22917.739,E2 -22917.739} C_VEL
LIN {X 0,Y 174.115,Z 334.367,A -85,B 0,C 180,E1 -22918.3,E2 -22918.3} C_VEL
LIN {X 0,Y 181.199,Z 346.338,A -85,B 0,C 180,E1 -22920.578,E2 -22920.578} C_VEL
LIN {X 0,Y 187.777,Z 359.058,A -85,B 0,C 180,E1 -22922.566,E2 -22922.566} C_VEL
LIN {X 0,Y 191.684,Z 368.126,A -85,B 0,C 180,E1 -22923.729,E2 -22923.729} C_VEL
LIN {X 0,Y 192.342,Z 369.991,A -85,B 0,C 180,E1 -22923.934,E2 -22923.934} C_VEL
LIN {X 0,Y 189.625,Z 429.501,A -85,B 0,C 180,E1 -22926.087,E2 -22926.087} C_VEL
LIN {X 0,Y 188.43,Z 443.194,A -85,B 0,C 180,E1 -22927.018,E2 -22927.018} C_VEL
LIN {X 0,Y 186.725,Z 456.05,A -85,B 0,C 180,E1 -22928.327,E2 -22928.327} C_VEL
LIN {X 0,Y 184.482,Z 467.811,A -85,B 0,C 180,E1 -22929.95,E2 -22929.95} C_VEL
LIN {X 0,Y 181.803,Z 479.152,A -85,B 0,C 180,E1 -22931.986,E2 -22931.986} C_VEL
LIN {X 0,Y 179.318,Z 489.331,A -85,B 0,C 180,E1 -22934.369,E2 -22934.369} C_VEL
LIN {X 0,Y 176.578,Z 499.301,A -85,B 0,C 180,E1 -22937.356,E2 -22937.356} C_VEL
LIN {X 0,Y 174.115,Z 508.075,A -85,B 0,C 180,E1 -22940.709,E2 -22940.709} C_VEL
LIN {X 0,Y 172.155,Z 515.096,A -85,B 0,C 180,E1 -22944.143,E2 -22944.143} C_VEL
LIN {X 0,Y 170.777,Z 520.7,A -85,B 0,C 180,E1 -22947.642,E2 -22947.642} C_VEL
LIN {X 0,Y 169.782,Z 525.124,A -85,B 0,C 180,E1 -22951.187,E2 -22951.187} C_VEL
LIN {X 0,Y 169.316,Z 528.657,A -85,B 0,C 180,E1 -22955.004,E2 -22955.004} C_VEL
LIN {X 0,Y 168.813,Z 531.444,A -85,B 0,C 180,E1 -22959.587,E2 -22959.587} C_VEL
LIN {X 0,Y 168.869,Z 532.318,A -85,B 0,C 180,E1 -22962.011,E2 -22962.011} C_VEL
LIN {X 0,Y 169.167,Z 532.75,A -85,B 0,C 180,E1 -22964.435,E2 -22964.435} C_VEL
LIN {X 0,Y 169.922,Z 532.697,A -85,B 0,C 180,E1 -22967.959,E2 -22967.959} C_VEL
LIN {X 0,Y 171.107,Z 531.684,A -85,B 0,C 180,E1 -22971.696,E2 -22971.696} C_VEL
LIN {X 0,Y 172.212,Z 530.472,A -85,B 0,C 180,E1 -22974.086,E2 -22974.086} C_VEL
LIN {X 0,Y 174.353,Z 527.938,A -85,B 0,C 180,E1 -22977.527,E2 -22977.527} C_VEL
LIN {X 0,Y 177.12,Z 524.201,A -85,B 0,C 180,E1 -22981.054,E2 -22981.054} C_VEL
LIN {X 0,Y 180.359,Z 519.37,A -85,B 0,C 180,E1 -22984.404,E2 -22984.404} C_VEL
LIN {X 0,Y 184.23,Z 513.223,A -85,B 0,C 180,E1 -22987.617,E2 -22987.617} C_VEL
LIN {X 0,Y 188.625,Z 505.528,A -85,B 0,C 180,E1 -22990.696,E2 -22990.696} C_VEL
LIN {X 0,Y 192.831,Z 497.351,A -85,B 0,C 180,E1 -22993.204,E2 -22993.204} C_VEL
LIN {X 0,Y 197.084,Z 487.838,A -85,B 0,C 180,E1 -22995.496,E2 -22995.496} C_VEL
LIN {X 0,Y 201.136,Z 476.928,A -85,B 0,C 180,E1 -22997.574,E2 -22997.574} C_VEL
LIN {X 0,Y 204.524,Z 466.295,A -85,B 0,C 180,E1 -22999.111,E2 -22999.111} C_VEL
LIN {X 0,Y 207.698,Z 453.366,A -85,B 0,C 180,E1 -23000.527,E2 -23000.527} C_VEL
LIN {X 0,Y 209.999,Z 440.536,A -85,B 0,C 180,E1 -23001.537,E2 -23001.537} C_VEL
LIN {X 0,Y 211.474,Z 428.246,A -85,B 0,C 180,E1 -23002.158,E2 -23002.158} C_VEL
LIN {X 0,Y 214.006,Z 391.247,A -85,B 0,C 180,E1 -23003.276,E2 -23003.276} C_VEL
LIN {X 0,Y 209.023,Z 380.827,A -85,B 0,C 180,E1 -23005.359,E2 -23005.359} C_VEL
LIN {X 0,Y 202.899,Z 370.544,A -85,B 0,C 180,E1 -23008.06,E2 -23008.06} C_VEL
LIN {X 0,Y 197.574,Z 362.538,A -85,B 0,C 180,E1 -23010.645,E2 -23010.645} C_VEL
LIN {X 0,Y 192.383,Z 355.162,A -85,B 0,C 180,E1 -23013.471,E2 -23013.471} C_VEL
LIN {X 0,Y 188.821,Z 350.522,A -85,B 0,C 180,E1 -23015.621,E2 -23015.621} C_VEL
LIN {X 0,Y 186.104,Z 347.132,A -85,B 0,C 180,E1 -23017.409,E2 -23017.409} C_VEL
LIN {X 0,Y 185.099,Z 345.71,A -85,B 0,C 180,E1 -23018.126,E2 -23018.126} C_VEL
LIN {X 0,Y 182.428,Z 342.89,A -85,B 0,C 180,E1 -23020.081,E2 -23020.081} C_VEL
LIN {X 0,Y 181.125,Z 340.599,A -85,B 0,C 180,E1 -23021.201,E2 -23021.201} C_VEL
LIN {X 0,Y 178.364,Z 338.271,A -85,B 0,C 180,E1 -23023.549,E2 -23023.549} C_VEL
LIN {X 0,Y 176.907,Z 335.547,A -85,B 0,C 180,E1 -23025.109,E2 -23025.109} C_VEL
LIN {X 0,Y 176.743,Z 335.054,A -85,B 0,C 180,E1 -23025.316,E2 -23025.316} C_VEL
LIN {X 0,Y 174.049,Z 333.472,A -85,B 0,C 180,E1 -23028.205,E2 -23028.205} C_VEL
LIN {X 0,Y 172.403,Z 330.952,A -85,B 0,C 180,E1 -23030.546,E2 -23030.546} C_VEL
LIN {X 0,Y 171.896,Z 329.071,A -85,B 0,C 180,E1 -23031.625,E2 -23031.625} C_VEL
LIN {X 0,Y 172.103,Z 329.032,A -85,B 0,C 180,E1 -23037.66,E2 -23037.66} C_VEL
LIN {X 0,Y 172.333,Z 329.015,A -85,B 0,C 180,E1 -23040.001,E2 -23040.001} C_VEL
LIN {X 0,Y 171.824,Z 329.078,A -85,B 0,C 180,E1 -23044.693,E2 -23044.693} C_VEL
LIN {X 0,Y 171.89,Z 329.071,A -85,B 0,C 180,E1 -23049.413,E2 -23049.413} C_VEL
LIN {X 0,Y 171.58,Z 329.108,A -85,B 0,C 180,E1 -23054.227,E2 -23054.227} C_VEL
LIN {X 0,Y 171.59,Z 329.28,A -85,B 0,C 180,E1 -23057.582,E2 -23057.582} C_VEL
LIN {X 0,Y 172.628,Z 332.072,A -85,B 0,C 180,E1 -23059.458,E2 -23059.458} C_VEL
LIN {X 0,Y 174.777,Z 334.304,A -85,B 0,C 180,E1 -23062.222,E2 -23062.222} C_VEL
LIN {X 0,Y 176.747,Z 335.479,A -85,B 0,C 180,E1 -23064.276,E2 -23064.276} C_VEL
LIN {X 0,Y 178.215,Z 338.27,A -85,B 0,C 180,E1 -23065.866,E2 -23065.866} C_VEL
LIN {X 0,Y 180.761,Z 341.14,A -85,B 0,C 180,E1 -23068.127,E2 -23068.127} C_VEL
LIN {X 0,Y 182.624,Z 343.384,A -85,B 0,C 180,E1 -23069.633,E2 -23069.633} C_VEL
LIN {X 0,Y 185.571,Z 347.721,A -85,B 0,C 180,E1 -23071.861,E2 -23071.861} C_VEL
LIN {X 0,Y 187.384,Z 350.287,A -85,B 0,C 180,E1 -23073.111,E2 -23073.111} C_VEL
LIN {X 0,Y 190.961,Z 355.858,A -85,B 0,C 180,E1 -23075.417,E2 -23075.417} C_VEL
LIN {X 0,Y 194.538,Z 361.651,A -85,B 0,C 180,E1 -23077.513,E2 -23077.513} C_VEL
LIN {X 0,Y 199.394,Z 369.878,A -85,B 0,C 180,E1 -23080.089,E2 -23080.089} C_VEL
LIN {X 0,Y 205.287,Z 381.288,A -85,B 0,C 180,E1 -23082.941,E2 -23082.941} C_VEL
LIN {X 0,Y 210.276,Z 392.494,A -85,B 0,C 180,E1 -23085.186,E2 -23085.186} C_VEL
LIN {X 0,Y 213.39,Z 400.176,A -85,B 0,C 180,E1 -23086.519,E2 -23086.519} C_VEL
LIN {X 0,Y 213.419,Z 403.24,A -85,B 0,C 180,E1 -23086.678,E2 -23086.678} C_VEL
LIN {X 0,Y 210.76,Z 441.566,A -85,B 0,C 180,E1 -23087.875,E2 -23087.875} C_VEL
LIN {X 0,Y 208.852,Z 454.872,A -85,B 0,C 180,E1 -23088.589,E2 -23088.589} C_VEL
LIN {X 0,Y 206.009,Z 467.733,A -85,B 0,C 180,E1 -23089.595,E2 -23089.595} C_VEL
LIN {X 0,Y 202.69,Z 479.163,A -85,B 0,C 180,E1 -23090.844,E2 -23090.844} C_VEL
LIN {X 0,Y 200.418,Z 484.359,A -85,B 0,C 180,E1 -23091.403,E2 -23091.403} C_VEL
LIN {X 0,Y 195.253,Z 492.442,A -85,B 0,C 180,E1 -23092.155,E2 -23092.155} C_VEL
LIN {X 0,Y 189.888,Z 500.039,A -85,B 0,C 180,E1 -23093.122,E2 -23093.122} C_VEL
LIN {X 0,Y 187.339,Z 504.412,A -85,B 0,C 180,E1 -23094.016,E2 -23094.016} C_VEL
LIN {X 0,Y 183.283,Z 512.425,A -85,B 0,C 180,E1 -23096.22,E2 -23096.22} C_VEL
LIN {X 0,Y 178.385,Z 520.889,A -85,B 0,C 180,E1 -23099.191,E2 -23099.191} C_VEL
LIN {X 0,Y 174.174,Z 527.705,A -85,B 0,C 180,E1 -23102.353,E2 -23102.353} C_VEL
LIN {X 0,Y 170.676,Z 533.179,A -85,B 0,C 180,E1 -23105.683,E2 -23105.683} C_VEL
LIN {X 0,Y 167.635,Z 537.492,A -85,B 0,C 180,E1 -23109.123,E2 -23109.123} C_VEL
LIN {X 0,Y 165.146,Z 540.759,A -85,B 0,C 180,E1 -23112.668,E2 -23112.668} C_VEL
LIN {X 0,Y 163.098,Z 543.654,A -85,B 0,C 180,E1 -23117.557,E2 -23117.557} C_VEL
LIN {X 0,Y 162.433,Z 544.486,A -85,B 0,C 180,E1 -23120.033,E2 -23120.033} C_VEL
LIN {X 0,Y 161.851,Z 544.959,A -85,B 0,C 180,E1 -23125.017,E2 -23125.017} C_VEL
LIN {X 0,Y 161.867,Z 544.624,A -85,B 0,C 180,E1 -23127.511,E2 -23127.511} C_VEL
LIN {X 0,Y 162.046,Z 543.889,A -85,B 0,C 180,E1 -23129.999,E2 -23129.999} C_VEL
LIN {X 0,Y 161.883,Z 542.329,A -85,B 0,C 180,E1 -23133.103,E2 -23133.103} C_VEL
LIN {X 0,Y 162.069,Z 539.039,A -85,B 0,C 180,E1 -23137.474,E2 -23137.474} C_VEL
LIN {X 0,Y 162.606,Z 535.057,A -85,B 0,C 180,E1 -23141.214,E2 -23141.214} C_VEL
LIN {X 0,Y 163.922,Z 528.908,A -85,B 0,C 180,E1 -23145.542,E2 -23145.542} C_VEL
LIN {X 0,Y 165.803,Z 522.177,A -85,B 0,C 180,E1 -23149.177,E2 -23149.177} C_VEL
LIN {X 0,Y 168.149,Z 514.055,A -85,B 0,C 180,E1 -23152.635,E2 -23152.635} C_VEL
LIN {X 0,Y 170.533,Z 505.165,A -85,B 0,C 180,E1 -23155.639,E2 -23155.639} C_VEL
LIN {X 0,Y 173.493,Z 494.514,A -85,B 0,C 180,E1 -23158.422,E2 -23158.422} C_VEL
LIN {X 0,Y 176.136,Z 483.944,A -85,B 0,C 180,E1 -23160.579,E2 -23160.579} C_VEL
LIN {X 0,Y 178.675,Z 472.262,A -85,B 0,C 180,E1 -23162.405,E2 -23162.405} C_VEL
LIN {X 0,Y 180.82,Z 460.102,A -85,B 0,C 180,E1 -23163.798,E2 -23163.798} C_VEL
LIN {X 0,Y 182.53,Z 446.859,A -85,B 0,C 180,E1 -23164.856,E2 -23164.856} C_VEL
LIN {X 0,Y 183.442,Z 433.95,A -85,B 0,C 180,E1 -23165.494,E2 -23165.494} C_VEL
LIN {X 0,Y 185.371,Z 393.296,A -85,B 0,C 180,E1 -23166.957,E2 -23166.957} C_VEL
LIN {X 0,Y 183.415,Z 372.878,A -85,B 0,C 180,E1 -23168.286,E2 -23168.286} C_VEL
LIN {X 0,Y 177.323,Z 356.938,A -85,B 0,C 180,E1 -23170.384,E2 -23170.384} C_VEL
LIN {X 0,Y 171.774,Z 344.774,A -85,B 0,C 180,E1 -23172.352,E2 -23172.352} C_VEL
LIN {X 0,Y 166.702,Z 335.454,A -85,B 0,C 180,E1 -23174.216,E2 -23174.216} C_VEL
LIN {X 0,Y 164.668,Z 331.553,A -85,B 0,C 180,E1 -23175.019,E2 -23175.019} C_VEL
LIN {X 0,Y 164.277,Z 330.025,A -85,B 0,C 180,E1 -23176.191,E2 -23176.191} C_VEL
LIN {X 0,Y 164.294,Z 330.022,A -85,B 0,C 180,E1 -23180.351,E2 -23180.351} C_VEL
LIN {X 0,Y 164.328,Z 330.019,A -85,B 0,C 180,E1 -23186.221,E2 -23186.221} C_VEL
LIN {X 0,Y 164.404,Z 330.009,A -85,B 0,C 180,E1 -23189.137,E2 -23189.137} C_VEL
LIN {X 0,Y 164.415,Z 330.004,A -85,B 0,C 180,E1 -23194.693,E2 -23194.693} C_VEL
LIN {X 0,Y 164.482,Z 329.996,A -85,B 0,C 180,E1 -23200.05,E2 -23200.05} C_VEL
LIN {X 0,Y 164.523,Z 329.988,A -85,B 0,C 180,E1 -23205.149,E2 -23205.149} C_VEL
LIN {X 0,Y 164.799,Z 329.934,A -85,B 0,C 180,E1 -23210.178,E2 -23210.178} C_VEL
LIN {X 0,Y 164.847,Z 329.948,A -85,B 0,C 180,E1 -23212.651,E2 -23212.651} C_VEL
LIN {X 0,Y 165.046,Z 329.905,A -85,B 0,C 180,E1 -23217.559,E2 -23217.559} C_VEL
LIN {X 0,Y 165.29,Z 329.868,A -85,B 0,C 180,E1 -23219.999,E2 -23219.999} C_VEL
LIN {X 0,Y 164.755,Z 329.962,A -85,B 0,C 180,E1 -23224.894,E2 -23224.894} C_VEL
LIN {X 0,Y 164.822,Z 329.94,A -85,B 0,C 180,E1 -23227.349,E2 -23227.349} C_VEL
LIN {X 0,Y 164.699,Z 329.944,A -85,B 0,C 180,E1 -23231.059,E2 -23231.059} C_VEL
LIN {X 0,Y 164.479,Z 329.988,A -85,B 0,C 180,E1 -23237.403,E2 -23237.403} C_VEL
LIN {X 0,Y 164.469,Z 329.97,A -85,B 0,C 180,E1 -23239.989,E2 -23239.989} C_VEL
LIN {X 0,Y 164.382,Z 330.008,A -85,B 0,C 180,E1 -23246.128,E2 -23246.128} C_VEL
LIN {X 0,Y 164.372,Z 329.987,A -85,B 0,C 180,E1 -23251.228,E2 -23251.228} C_VEL
LIN {X 0,Y 164.291,Z 330.008,A -85,B 0,C 180,E1 -23256.79,E2 -23256.79} C_VEL
LIN {X 0,Y 164.287,Z 330.002,A -85,B 0,C 180,E1 -23259.917,E2 -23259.917} C_VEL
LIN {X 0,Y 164.276,Z 330.018,A -85,B 0,C 180,E1 -23263.342,E2 -23263.342} C_VEL
LIN {X 0,Y 164.257,Z 330.009,A -85,B 0,C 180,E1 -23266.799,E2 -23266.799} C_VEL
LIN {X 0,Y 164.286,Z 330.015,A -85,B 0,C 180,E1 -23270.355,E2 -23270.355} C_VEL
LIN {X 0,Y 164.369,Z 330.009,A -85,B 0,C 180,E1 -23275.373,E2 -23275.373} C_VEL
LIN {X 0,Y 165.366,Z 332.854,A -85,B 0,C 180,E1 -23275.847,E2 -23275.847} C_VEL
LIN {X 0,Y 167.157,Z 335.126,A -85,B 0,C 180,E1 -23276.485,E2 -23276.485} C_VEL
LIN {X 0,Y 175.193,Z 348.599,A -85,B 0,C 180,E1 -23279.29,E2 -23279.29} C_VEL
LIN {X 0,Y 181.994,Z 361.61,A -85,B 0,C 180,E1 -23281.478,E2 -23281.478} C_VEL
LIN {X 0,Y 186.13,Z 371.292,A -85,B 0,C 180,E1 -23282.789,E2 -23282.789} C_VEL
LIN {X 0,Y 186.303,Z 373.719,A -85,B 0,C 180,E1 -23282.934,E2 -23282.934} C_VEL
LIN {X 0,Y 183.523,Z 429.452,A -85,B 0,C 180,E1 -23284.976,E2 -23284.976} C_VEL
LIN {X 0,Y 182.32,Z 442.85,A -85,B 0,C 180,E1 -23285.899,E2 -23285.899} C_VEL
LIN {X 0,Y 180.544,Z 455.901,A -85,B 0,C 180,E1 -23287.243,E2 -23287.243} C_VEL
LIN {X 0,Y 178.206,Z 467.755,A -85,B 0,C 180,E1 -23288.909,E2 -23288.909} C_VEL
LIN {X 0,Y 175.403,Z 479.157,A -85,B 0,C 180,E1 -23291.002,E2 -23291.002} C_VEL
LIN {X 0,Y 172.798,Z 489.388,A -85,B 0,C 180,E1 -23293.46,E2 -23293.46} C_VEL
LIN {X 0,Y 170.164,Z 498.588,A -85,B 0,C 180,E1 -23296.263,E2 -23296.263} C_VEL
LIN {X 0,Y 167.522,Z 507.525,A -85,B 0,C 180,E1 -23299.73,E2 -23299.73} C_VEL
LIN {X 0,Y 165.39,Z 514.73,A -85,B 0,C 180,E1 -23303.29,E2 -23303.29} C_VEL
LIN {X 0,Y 164.095,Z 519.586,A -85,B 0,C 180,E1 -23306.318,E2 -23306.318} C_VEL
LIN {X 0,Y 162.894,Z 524.32,A -85,B 0,C 180,E1 -23310.001,E2 -23310.001} C_VEL
LIN {X 0,Y 162.508,Z 526.866,A -85,B 0,C 180,E1 -23312.48,E2 -23312.48} C_VEL
LIN {X 0,Y 162.215,Z 528.92,A -85,B 0,C 180,E1 -23314.972,E2 -23314.972} C_VEL
LIN {X 0,Y 161.852,Z 530.575,A -85,B 0,C 180,E1 -23317.486,E2 -23317.486} C_VEL
LIN {X 0,Y 161.726,Z 531.825,A -85,B 0,C 180,E1 -23320.011,E2 -23320.011} C_VEL
LIN {X 0,Y 161.81,Z 532.637,A -85,B 0,C 180,E1 -23322.544,E2 -23322.544} C_VEL
LIN {X 0,Y 162.184,Z 533.034,A -85,B 0,C 180,E1 -23325.071,E2 -23325.071} C_VEL
LIN {X 0,Y 162.9,Z 532.989,A -85,B 0,C 180,E1 -23328.353,E2 -23328.353} C_VEL
LIN {X 0,Y 164.351,Z 531.839,A -85,B 0,C 180,E1 -23332.636,E2 -23332.636} C_VEL
LIN {X 0,Y 165.593,Z 530.594,A -85,B 0,C 180,E1 -23335.114,E2 -23335.114} C_VEL
LIN {X 0,Y 167.642,Z 528.316,A -85,B 0,C 180,E1 -23338.313,E2 -23338.313} C_VEL
LIN {X 0,Y 170.886,Z 524.179,A -85,B 0,C 180,E1 -23342.321,E2 -23342.321} C_VEL
LIN {X 0,Y 174.357,Z 519.308,A -85,B 0,C 180,E1 -23345.736,E2 -23345.736} C_VEL
LIN {X 0,Y 178.504,Z 513.035,A -85,B 0,C 180,E1 -23349.047,E2 -23349.047} C_VEL
LIN {X 0,Y 183.158,Z 505.203,A -85,B 0,C 180,E1 -23352.183,E2 -23352.183} C_VEL
LIN {X 0,Y 187.743,Z 496.572,A -85,B 0,C 180,E1 -23354.814,E2 -23354.814} C_VEL
LIN {X 0,Y 192.49,Z 486.144,A -85,B 0,C 180,E1 -23357.29,E2 -23357.29} C_VEL
LIN {X 0,Y 196.29,Z 476.138,A -85,B 0,C 180,E1 -23359.14,E2 -23359.14} C_VEL
LIN {X 0,Y 200.26,Z 463.688,A -85,B 0,C 180,E1 -23360.862,E2 -23360.862} C_VEL
LIN {X 0,Y 203.069,Z 452.157,A -85,B 0,C 180,E1 -23362.08,E2 -23362.08} C_VEL
LIN {X 0,Y 205.341,Z 439.236,A -85,B 0,C 180,E1 -23363.062,E2 -23363.062} C_VEL
LIN {X 0,Y 206.829,Z 426.874,A -85,B 0,C 180,E1 -23363.634,E2 -23363.634} C_VEL
LIN {X 0,Y 209.13,Z 393.823,A -85,B 0,C 180,E1 -23364.645,E2 -23364.645} C_VEL
LIN {X 0,Y 204.952,Z 385.036,A -85,B 0,C 180,E1 -23366.505,E2 -23366.505} C_VEL
LIN {X 0,Y 199.003,Z 375.019,A -85,B 0,C 180,E1 -23369.29,E2 -23369.29} C_VEL
LIN {X 0,Y 194.448,Z 367.991,A -85,B 0,C 180,E1 -23371.645,E2 -23371.645} C_VEL
LIN {X 0,Y 189.547,Z 360.892,A -85,B 0,C 180,E1 -23374.467,E2 -23374.467} C_VEL
LIN {X 0,Y 186.325,Z 356.576,A -85,B 0,C 180,E1 -23376.522,E2 -23376.522} C_VEL
LIN {X 0,Y 183.499,Z 352.684,A -85,B 0,C 180,E1 -23378.516,E2 -23378.516} C_VEL
LIN {X 0,Y 180.24,Z 348.944,A -85,B 0,C 180,E1 -23381.028,E2 -23381.028} C_VEL
LIN {X 0,Y 179.149,Z 347.124,A -85,B 0,C 180,E1 -23382.005,E2 -23382.005} C_VEL
LIN {X 0,Y 176.439,Z 344.502,A -85,B 0,C 180,E1 -23384.478,E2 -23384.478} C_VEL
LIN {X 0,Y 175.053,Z 341.855,A -85,B 0,C 180,E1 -23386.062,E2 -23386.062} C_VEL
LIN {X 0,Y 172.474,Z 339.993,A -85,B 0,C 180,E1 -23389.034,E2 -23389.034} C_VEL
LIN {X 0,Y 170.853,Z 337.158,A -85,B 0,C 180,E1 -23391.574,E2 -23391.574} C_VEL
LIN {X 0,Y 170.497,Z 336.028,A -85,B 0,C 180,E1 -23392.302,E2 -23392.302} C_VEL
LIN {X 0,Y 167.903,Z 334.768,A -85,B 0,C 180,E1 -23397.602,E2 -23397.602} C_VEL
LIN {X 0,Y 167.254,Z 333.944,A -85,B 0,C 180,E1 -23400.001,E2 -23400.001} C_VEL
LIN {X 0,Y 166.888,Z 334.119,A -85,B 0,C 180,E1 -23407.867,E2 -23407.867} C_VEL
LIN {X 0,Y 170.279,Z 336.263,A -85,B 0,C 180,E1 -23416.948,E2 -23416.948} C_VEL
LIN {X 0,Y 171.66,Z 339.396,A -85,B 0,C 180,E1 -23419.421,E2 -23419.421} C_VEL
LIN {X 0,Y 174.085,Z 341.517,A -85,B 0,C 180,E1 -23422.475,E2 -23422.475} C_VEL
LIN {X 0,Y 175.073,Z 342.171,A -85,B 0,C 180,E1 -23423.535,E2 -23423.535} C_VEL
LIN {X 0,Y 176.874,Z 345.256,A -85,B 0,C 180,E1 -23425.52,E2 -23425.52} C_VEL
LIN {X 0,Y 180.251,Z 349.092,A -85,B 0,C 180,E1 -23428.531,E2 -23428.531} C_VEL
LIN {X 0,Y 183.141,Z 353.688,A -85,B 0,C 180,E1 -23430.882,E2 -23430.882} C_VEL
LIN {X 0,Y 184.886,Z 356.174,A -85,B 0,C 180,E1 -23432.153,E2 -23432.153} C_VEL
LIN {X 0,Y 188.431,Z 361.906,A -85,B 0,C 180,E1 -23434.568,E2 -23434.568} C_VEL
LIN {X 0,Y 191.813,Z 367.569,A -85,B 0,C 180,E1 -23436.657,E2 -23436.657} C_VEL
LIN {X 0,Y 196.697,Z 376.284,A -85,B 0,C 180,E1 -23439.389,E2 -23439.389} C_VEL
LIN {X 0,Y 202.067,Z 387.019,A -85,B 0,C 180,E1 -23442.115,E2 -23442.115} C_VEL
LIN {X 0,Y 207.627,Z 400.209,A -85,B 0,C 180,E1 -23444.743,E2 -23444.743} C_VEL
LIN {X 0,Y 208.687,Z 403.35,A -85,B 0,C 180,E1 -23445.244,E2 -23445.244} C_VEL
LIN {X 0,Y 205.943,Z 441.318,A -85,B 0,C 180,E1 -23446.441,E2 -23446.441} C_VEL
LIN {X 0,Y 203.908,Z 454.986,A -85,B 0,C 180,E1 -23447.184,E2 -23447.184} C_VEL
LIN {X 0,Y 200.953,Z 467.716,A -85,B 0,C 180,E1 -23448.188,E2 -23448.188} C_VEL
LIN {X 0,Y 197.426,Z 479.403,A -85,B 0,C 180,E1 -23449.487,E2 -23449.487} C_VEL
LIN {X 0,Y 193.418,Z 490.641,A -85,B 0,C 180,E1 -23451.185,E2 -23451.185} C_VEL
LIN {X 0,Y 189.027,Z 500.823,A -85,B 0,C 180,E1 -23453.163,E2 -23453.163} C_VEL
LIN {X 0,Y 187.339,Z 504.412,A -85,B 0,C 180,E1 -23454.016,E2 -23454.016} C_VEL
LIN {X 0,Y 184.705,Z 508.671,A -85,B 0,C 180,E1 -23454.994,E2 -23454.994} C_VEL
LIN {X 0,Y 178.836,Z 515.179,A -85,B 0,C 180,E1 -23456.451,E2 -23456.451} C_VEL
LIN {X 0,Y 172.854,Z 521.127,A -85,B 0,C 180,E1 -23458.15,E2 -23458.15} C_VEL
LIN {X 0,Y 170.103,Z 524.413,A -85,B 0,C 180,E1 -23459.503,E2 -23459.503} C_VEL
LIN {X 0,Y 165.793,Z 530.866,A -85,B 0,C 180,E1 -23463.082,E2 -23463.082} C_VEL
LIN {X 0,Y 161.951,Z 536.142,A -85,B 0,C 180,E1 -23467.01,E2 -23467.01} C_VEL
LIN {X 0,Y 159.198,Z 539.686,A -85,B 0,C 180,E1 -23470.664,E2 -23470.664} C_VEL
LIN {X 0,Y 157.056,Z 542.248,A -85,B 0,C 180,E1 -23474.425,E2 -23474.425} C_VEL
LIN {X 0,Y 156.125,Z 543.469,A -85,B 0,C 180,E1 -23476.992,E2 -23476.992} C_VEL
LIN {X 0,Y 154.97,Z 544.659,A -85,B 0,C 180,E1 -23482.18,E2 -23482.18} C_VEL
LIN {X 0,Y 154.777,Z 544.323,A -85,B 0,C 180,E1 -23487.397,E2 -23487.397} C_VEL
LIN {X 0,Y 154.951,Z 543.539,A -85,B 0,C 180,E1 -23489.999,E2 -23489.999} C_VEL
LIN {X 0,Y 154.815,Z 542.15,A -85,B 0,C 180,E1 -23492.893,E2 -23492.893} C_VEL
LIN {X 0,Y 154.901,Z 539.686,A -85,B 0,C 180,E1 -23496.512,E2 -23496.512} C_VEL
LIN {X 0,Y 155.341,Z 536.013,A -85,B 0,C 180,E1 -23500.425,E2 -23500.425} C_VEL
LIN {X 0,Y 156.297,Z 531.201,A -85,B 0,C 180,E1 -23504.317,E2 -23504.317} C_VEL
LIN {X 0,Y 158.004,Z 525.118,A -85,B 0,C 180,E1 -23508.14,E2 -23508.14} C_VEL
LIN {X 0,Y 160.335,Z 517.534,A -85,B 0,C 180,E1 -23511.874,E2 -23511.874} C_VEL
LIN {X 0,Y 162.636,Z 509.543,A -85,B 0,C 180,E1 -23515.006,E2 -23515.006} C_VEL
LIN {X 0,Y 165.359,Z 500.287,A -85,B 0,C 180,E1 -23517.872,E2 -23517.872} C_VEL
LIN {X 0,Y 168.244,Z 489.746,A -85,B 0,C 180,E1 -23520.429,E2 -23520.429} C_VEL
LIN {X 0,Y 171.179,Z 478.039,A -85,B 0,C 180,E1 -23522.605,E2 -23522.605} C_VEL
LIN {X 0,Y 173.535,Z 466.695,A -85,B 0,C 180,E1 -23524.188,E2 -23524.188} C_VEL
LIN {X 0,Y 175.539,Z 453.893,A -85,B 0,C 180,E1 -23525.487,E2 -23525.487} C_VEL
LIN {X 0,Y 176.964,Z 440.534,A -85,B 0,C 180,E1 -23526.385,E2 -23526.385} C_VEL
LIN {X 0,Y 179.394,Z 393.968,A -85,B 0,C 180,E1 -23528.141,E2 -23528.141} C_VEL
LIN {X 0,Y 177.603,Z 375.015,A -85,B 0,C 180,E1 -23529.438,E2 -23529.438} C_VEL
LIN {X 0,Y 171.483,Z 358.852,A -85,B 0,C 180,E1 -23531.696,E2 -23531.696} C_VEL
LIN {X 0,Y 165.164,Z 345.402,A -85,B 0,C 180,E1 -23534.105,E2 -23534.105} C_VEL
LIN {X 0,Y 159.556,Z 335.38,A -85,B 0,C 180,E1 -23536.362,E2 -23536.362} C_VEL
LIN {X 0,Y 157.657,Z 332.649,A -85,B 0,C 180,E1 -23537.142,E2 -23537.142} C_VEL
LIN {X 0,Y 157.228,Z 331.177,A -85,B 0,C 180,E1 -23537.383,E2 -23537.383} C_VEL
LIN {X 0,Y 157.191,Z 330.906,A -85,B 0,C 180,E1 -23537.882,E2 -23537.882} C_VEL
LIN {X 0,Y 157.266,Z 330.9,A -85,B 0,C 180,E1 -23543.55,E2 -23543.55} C_VEL
LIN {X 0,Y 157.299,Z 330.892,A -85,B 0,C 180,E1 -23548.09,E2 -23548.09} C_VEL
LIN {X 0,Y 157.32,Z 330.89,A -85,B 0,C 180,E1 -23553.465,E2 -23553.465} C_VEL
LIN {X 0,Y 157.392,Z 330.881,A -85,B 0,C 180,E1 -23559.666,E2 -23559.666} C_VEL
LIN {X 0,Y 157.452,Z 330.872,A -85,B 0,C 180,E1 -23564.465,E2 -23564.465} C_VEL
LIN {X 0,Y 157.723,Z 330.811,A -85,B 0,C 180,E1 -23569.732,E2 -23569.732} C_VEL
LIN {X 0,Y 157.804,Z 330.824,A -85,B 0,C 180,E1 -23572.321,E2 -23572.321} C_VEL
LIN {X 0,Y 158.252,Z 330.743,A -85,B 0,C 180,E1 -23579.999,E2 -23579.999} C_VEL
LIN {X 0,Y 157.76,Z 330.816,A -85,B 0,C 180,E1 -23587.68,E2 -23587.68} C_VEL
LIN {X 0,Y 157.633,Z 330.824,A -85,B 0,C 180,E1 -23591.235,E2 -23591.235} C_VEL
LIN {X 0,Y 157.45,Z 330.872,A -85,B 0,C 180,E1 -23595.534,E2 -23595.534} C_VEL
LIN {X 0,Y 157.364,Z 330.855,A -85,B 0,C 180,E1 -23600.933,E2 -23600.933} C_VEL
LIN {X 0,Y 157.306,Z 330.886,A -85,B 0,C 180,E1 -23606.681,E2 -23606.681} C_VEL
LIN {X 0,Y 157.272,Z 330.882,A -85,B 0,C 180,E1 -23612.428,E2 -23612.428} C_VEL
LIN {X 0,Y 157.264,Z 330.885,A -85,B 0,C 180,E1 -23616.45,E2 -23616.45} C_VEL
LIN {X 0,Y 157.189,Z 330.902,A -85,B 0,C 180,E1 -23622.117,E2 -23622.117} C_VEL
LIN {X 0,Y 157.186,Z 330.898,A -85,B 0,C 180,E1 -23627.883,E2 -23627.883} C_VEL
LIN {X 0,Y 157.236,Z 330.892,A -85,B 0,C 180,E1 -23633.167,E2 -23633.167} C_VEL
LIN {X 0,Y 158.335,Z 333.843,A -85,B 0,C 180,E1 -23633.744,E2 -23633.744} C_VEL
LIN {X 0,Y 160.351,Z 336.364,A -85,B 0,C 180,E1 -23634.537,E2 -23634.537} C_VEL
LIN {X 0,Y 165.424,Z 344.46,A -85,B 0,C 180,E1 -23636.509,E2 -23636.509} C_VEL
LIN {X 0,Y 171.371,Z 354.697,A -85,B 0,C 180,E1 -23638.653,E2 -23638.653} C_VEL
LIN {X 0,Y 177.685,Z 367.394,A -85,B 0,C 180,E1 -23640.803,E2 -23640.803} C_VEL
LIN {X 0,Y 180.383,Z 373.882,A -85,B 0,C 180,E1 -23641.71,E2 -23641.71} C_VEL
LIN {X 0,Y 177.438,Z 430.099,A -85,B 0,C 180,E1 -23643.83,E2 -23643.83} C_VEL
LIN {X 0,Y 176.099,Z 444.018,A -85,B 0,C 180,E1 -23644.833,E2 -23644.833} C_VEL
LIN {X 0,Y 174.238,Z 456.768,A -85,B 0,C 180,E1 -23646.213,E2 -23646.213} C_VEL
LIN {X 0,Y 171.993,Z 467.698,A -85,B 0,C 180,E1 -23647.793,E2 -23647.793} C_VEL
LIN {X 0,Y 169.064,Z 479.16,A -85,B 0,C 180,E1 -23649.944,E2 -23649.944} C_VEL
LIN {X 0,Y 166.327,Z 489.441,A -85,B 0,C 180,E1 -23652.48,E2 -23652.48} C_VEL
LIN {X 0,Y 163.8,Z 497.862,A -85,B 0,C 180,E1 -23655.083,E2 -23655.083} C_VEL
LIN {X 0,Y 160.973,Z 506.977,A -85,B 0,C 180,E1 -23658.671,E2 -23658.671} C_VEL
LIN {X 0,Y 158.686,Z 514.322,A -85,B 0,C 180,E1 -23662.366,E2 -23662.366} C_VEL
LIN {X 0,Y 157.019,Z 520.211,A -85,B 0,C 180,E1 -23666.151,E2 -23666.151} C_VEL
LIN {X 0,Y 155.799,Z 524.869,A -85,B 0,C 180,E1 -23670.001,E2 -23670.001} C_VEL
LIN {X 0,Y 155.397,Z 527.346,A -85,B 0,C 180,E1 -23672.593,E2 -23672.593} C_VEL
LIN {X 0,Y 155.063,Z 529.368,A -85,B 0,C 180,E1 -23675.202,E2 -23675.202} C_VEL
LIN {X 0,Y 154.724,Z 530.989,A -85,B 0,C 180,E1 -23677.833,E2 -23677.833} C_VEL
LIN {X 0,Y 154.622,Z 532.196,A -85,B 0,C 180,E1 -23680.476,E2 -23680.476} C_VEL
LIN {X 0,Y 155.191,Z 533.32,A -85,B 0,C 180,E1 -23685.767,E2 -23685.767} C_VEL
LIN {X 0,Y 155.905,Z 533.273,A -85,B 0,C 180,E1 -23688.801,E2 -23688.801} C_VEL
LIN {X 0,Y 157.646,Z 531.995,A -85,B 0,C 180,E1 -23693.656,E2 -23693.656} C_VEL
LIN {X 0,Y 159.016,Z 530.716,A -85,B 0,C 180,E1 -23696.23,E2 -23696.23} C_VEL
LIN {X 0,Y 160.974,Z 528.688,A -85,B 0,C 180,E1 -23699.17,E2 -23699.17} C_VEL
LIN {X 0,Y 164.744,Z 524.16,A -85,B 0,C 180,E1 -23703.683,E2 -23703.683} C_VEL
LIN {X 0,Y 168.299,Z 519.472,A -85,B 0,C 180,E1 -23707.021,E2 -23707.021} C_VEL
LIN {X 0,Y 172.897,Z 512.854,A -85,B 0,C 180,E1 -23710.57,E2 -23710.57} C_VEL
LIN {X 0,Y 177.831,Z 504.875,A -85,B 0,C 180,E1 -23713.759,E2 -23713.759} C_VEL
LIN {X 0,Y 182.618,Z 496.149,A -85,B 0,C 180,E1 -23716.423,E2 -23716.423} C_VEL
LIN {X 0,Y 187.133,Z 486.642,A -85,B 0,C 180,E1 -23718.688,E2 -23718.688} C_VEL
LIN {X 0,Y 191.563,Z 475.435,A -85,B 0,C 180,E1 -23720.753,E2 -23720.753} C_VEL
LIN {X 0,Y 195.33,Z 463.999,A -85,B 0,C 180,E1 -23722.332,E2 -23722.332} C_VEL
LIN {X 0,Y 198.216,Z 452.571,A -85,B 0,C 180,E1 -23723.554,E2 -23723.554} C_VEL
LIN {X 0,Y 200.577,Z 439.783,A -85,B 0,C 180,E1 -23724.538,E2 -23724.538} C_VEL
LIN {X 0,Y 202.104,Z 427.712,A -85,B 0,C 180,E1 -23725.11,E2 -23725.11} C_VEL
LIN {X 0,Y 204.429,Z 396.647,A -85,B 0,C 180,E1 -23726.048,E2 -23726.048} C_VEL
LIN {X 0,Y 201.119,Z 389.56,A -85,B 0,C 180,E1 -23727.623,E2 -23727.623} C_VEL
LIN {X 0,Y 195.672,Z 380.169,A -85,B 0,C 180,E1 -23730.332,E2 -23730.332} C_VEL
LIN {X 0,Y 191.137,Z 373.011,A -85,B 0,C 180,E1 -23732.823,E2 -23732.823} C_VEL
LIN {X 0,Y 186.516,Z 366.217,A -85,B 0,C 180,E1 -23735.662,E2 -23735.662} C_VEL
LIN {X 0,Y 183.908,Z 362.594,A -85,B 0,C 180,E1 -23737.431,E2 -23737.431} C_VEL
LIN {X 0,Y 180.73,Z 358.304,A -85,B 0,C 180,E1 -23739.811,E2 -23739.811} C_VEL
LIN {X 0,Y 178.059,Z 354.916,A -85,B 0,C 180,E1 -23742.04,E2 -23742.04} C_VEL
LIN {X 0,Y 177.158,Z 353.576,A -85,B 0,C 180,E1 -23742.877,E2 -23742.877} C_VEL
LIN {X 0,Y 174.439,Z 350.538,A -85,B 0,C 180,E1 -23745.565,E2 -23745.565} C_VEL
LIN {X 0,Y 173.429,Z 348.614,A -85,B 0,C 180,E1 -23746.791,E2 -23746.791} C_VEL
LIN {X 0,Y 170.91,Z 346.465,A -85,B 0,C 180,E1 -23749.919,E2 -23749.919} C_VEL
LIN {X 0,Y 169.379,Z 343.439,A -85,B 0,C 180,E1 -23752.572,E2 -23752.572} C_VEL
LIN {X 0,Y 169.261,Z 342.995,A -85,B 0,C 180,E1 -23752.845,E2 -23752.845} C_VEL
LIN {X 0,Y 166.502,Z 341.28,A -85,B 0,C 180,E1 -23759.396,E2 -23759.396} C_VEL
LIN {X 0,Y 165.944,Z 340.847,A -85,B 0,C 180,E1 -23762.428,E2 -23762.428} C_VEL
LIN {X 0,Y 166.232,Z 341.392,A -85,B 0,C 180,E1 -23769.123,E2 -23769.123} C_VEL
LIN {X 0,Y 169.07,Z 343.323,A -85,B 0,C 180,E1 -23776.451,E2 -23776.451} C_VEL
LIN {X 0,Y 170.514,Z 346.377,A -85,B 0,C 180,E1 -23779.097,E2 -23779.097} C_VEL
LIN {X 0,Y 172.826,Z 348.394,A -85,B 0,C 180,E1 -23782.096,E2 -23782.096} C_VEL
LIN {X 0,Y 173.597,Z 349.118,A -85,B 0,C 180,E1 -23782.981,E2 -23782.981} C_VEL
LIN {X 0,Y 175.588,Z 352.241,A -85,B 0,C 180,E1 -23785.21,E2 -23785.21} C_VEL
LIN {X 0,Y 178.449,Z 355.869,A -85,B 0,C 180,E1 -23787.885,E2 -23787.885} C_VEL
LIN {X 0,Y 181.615,Z 360.694,A -85,B 0,C 180,E1 -23790.525,E2 -23790.525} C_VEL
LIN {X 0,Y 185.921,Z 367.9,A -85,B 0,C 180,E1 -23793.68,E2 -23793.68} C_VEL
LIN {X 0,Y 189.28,Z 373.788,A -85,B 0,C 180,E1 -23795.869,E2 -23795.869} C_VEL
LIN {X 0,Y 193.414,Z 381.423,A -85,B 0,C 180,E1 -23798.316,E2 -23798.316} C_VEL
LIN {X 0,Y 198.377,Z 391.649,A -85,B 0,C 180,E1 -23801,E2 -23801} C_VEL
LIN {X 0,Y 203.633,Z 404.614,A -85,B 0,C 180,E1 -23803.651,E2 -23803.651} C_VEL
LIN {X 0,Y 203.948,Z 405.387,A -85,B 0,C 180,E1 -23803.801,E2 -23803.801} C_VEL
LIN {X 0,Y 201.262,Z 441.129,A -85,B 0,C 180,E1 -23804.943,E2 -23804.943} C_VEL
LIN {X 0,Y 199.221,Z 454.363,A -85,B 0,C 180,E1 -23805.658,E2 -23805.658} C_VEL
LIN {X 0,Y 196.326,Z 466.705,A -85,B 0,C 180,E1 -23806.617,E2 -23806.617} C_VEL
LIN {X 0,Y 192.686,Z 478.534,A -85,B 0,C 180,E1 -23807.916,E2 -23807.916} C_VEL
LIN {X 0,Y 189.001,Z 488.614,A -85,B 0,C 180,E1 -23809.402,E2 -23809.402} C_VEL
LIN {X 0,Y 184.385,Z 499.113,A -85,B 0,C 180,E1 -23811.38,E2 -23811.38} C_VEL
LIN {X 0,Y 180.093,Z 507.706,A -85,B 0,C 180,E1 -23813.478,E2 -23813.478} C_VEL
LIN {X 0,Y 175.655,Z 515.641,A -85,B 0,C 180,E1 -23815.934,E2 -23815.934} C_VEL
LIN {X 0,Y 170.775,Z 523.443,A -85,B 0,C 180,E1 -23819.041,E2 -23819.041} C_VEL
LIN {X 0,Y 170.103,Z 524.413,A -85,B 0,C 180,E1 -23819.503,E2 -23819.503} C_VEL
LIN {X 0,Y 167.416,Z 527.523,A -85,B 0,C 180,E1 -23820.962,E2 -23820.962} C_VEL
LIN {X 0,Y 161.675,Z 532.067,A -85,B 0,C 180,E1 -23823.3,E2 -23823.3} C_VEL
LIN {X 0,Y 156.183,Z 535.919,A -85,B 0,C 180,E1 -23825.927,E2 -23825.927} C_VEL
LIN {X 0,Y 153.954,Z 537.872,A -85,B 0,C 180,E1 -23827.807,E2 -23827.807} C_VEL
LIN {X 0,Y 151.63,Z 540.505,A -85,B 0,C 180,E1 -23831.067,E2 -23831.067} C_VEL
LIN {X 0,Y 150.191,Z 542.094,A -85,B 0,C 180,E1 -23833.693,E2 -23833.693} C_VEL
LIN {X 0,Y 149.172,Z 543.272,A -85,B 0,C 180,E1 -23836.374,E2 -23836.374} C_VEL
LIN {X 0,Y 147.939,Z 544.406,A -85,B 0,C 180,E1 -23841.805,E2 -23841.805} C_VEL
LIN {X 0,Y 147.691,Z 544.404,A -85,B 0,C 180,E1 -23844.538,E2 -23844.538} C_VEL
LIN {X 0,Y 147.695,Z 543.861,A -85,B 0,C 180,E1 -23847.835,E2 -23847.835} C_VEL
LIN {X 0,Y 147.858,Z 543.188,A -85,B 0,C 180,E1 -23849.999,E2 -23849.999} C_VEL
LIN {X 0,Y 147.723,Z 541.936,A -85,B 0,C 180,E1 -23852.726,E2 -23852.726} C_VEL
LIN {X 0,Y 147.819,Z 539.255,A -85,B 0,C 180,E1 -23856.825,E2 -23856.825} C_VEL
LIN {X 0,Y 148.324,Z 535.527,A -85,B 0,C 180,E1 -23860.924,E2 -23860.924} C_VEL
LIN {X 0,Y 149.383,Z 530.655,A -85,B 0,C 180,E1 -23864.995,E2 -23864.995} C_VEL
LIN {X 0,Y 151.233,Z 524.506,A -85,B 0,C 180,E1 -23868.983,E2 -23868.983} C_VEL
LIN {X 0,Y 153.75,Z 516.85,A -85,B 0,C 180,E1 -23872.862,E2 -23872.862} C_VEL
LIN {X 0,Y 155.367,Z 511.168,A -85,B 0,C 180,E1 -23875.216,E2 -23875.216} C_VEL
LIN {X 0,Y 158.387,Z 501.447,A -85,B 0,C 180,E1 -23878.488,E2 -23878.488} C_VEL
LIN {X 0,Y 161.346,Z 491.274,A -85,B 0,C 180,E1 -23881.147,E2 -23881.147} C_VEL
LIN {X 0,Y 164.397,Z 479.974,A -85,B 0,C 180,E1 -23883.394,E2 -23883.394} C_VEL
LIN {X 0,Y 167.025,Z 468.259,A -85,B 0,C 180,E1 -23885.164,E2 -23885.164} C_VEL
LIN {X 0,Y 169.239,Z 455.559,A -85,B 0,C 180,E1 -23886.558,E2 -23886.558} C_VEL
LIN {X 0,Y 170.84,Z 442.01,A -85,B 0,C 180,E1 -23887.541,E2 -23887.541} C_VEL
LIN {X 0,Y 172.592,Z 413.183,A -85,B 0,C 180,E1 -23888.69,E2 -23888.69} C_VEL
LIN {X 0,Y 173.439,Z 394.456,A -85,B 0,C 180,E1 -23889.426,E2 -23889.426} C_VEL
LIN {X 0,Y 171.952,Z 377.438,A -85,B 0,C 180,E1 -23890.629,E2 -23890.629} C_VEL
LIN {X 0,Y 166.303,Z 362.276,A -85,B 0,C 180,E1 -23892.865,E2 -23892.865} C_VEL
LIN {X 0,Y 160.406,Z 349.555,A -85,B 0,C 180,E1 -23895.27,E2 -23895.27} C_VEL
LIN {X 0,Y 155.451,Z 340.491,A -85,B 0,C 180,E1 -23897.402,E2 -23897.402} C_VEL
LIN {X 0,Y 153.331,Z 337.294,A -85,B 0,C 180,E1 -23898.336,E2 -23898.336} C_VEL
LIN {X 0,Y 152.41,Z 336.164,A -85,B 0,C 180,E1 -23898.738,E2 -23898.738} C_VEL
LIN {X 0,Y 150.65,Z 333.644,A -85,B 0,C 180,E1 -23899.552,E2 -23899.552} C_VEL
LIN {X 0,Y 150.149,Z 331.783,A -85,B 0,C 180,E1 -23899.939,E2 -23899.939} C_VEL
LIN {X 0,Y 150.178,Z 331.78,A -85,B 0,C 180,E1 -23902.706,E2 -23902.706} C_VEL
LIN {X 0,Y 150.219,Z 331.776,A -85,B 0,C 180,E1 -23907.363,E2 -23907.363} C_VEL
LIN {X 0,Y 150.243,Z 331.773,A -85,B 0,C 180,E1 -23912.716,E2 -23912.716} C_VEL
LIN {X 0,Y 150.349,Z 331.756,A -85,B 0,C 180,E1 -23919.207,E2 -23919.207} C_VEL
LIN {X 0,Y 150.36,Z 331.756,A -85,B 0,C 180,E1 -23923.712,E2 -23923.712} C_VEL
LIN {X 0,Y 150.645,Z 331.689,A -85,B 0,C 180,E1 -23929.244,E2 -23929.244} C_VEL
LIN {X 0,Y 150.739,Z 331.699,A -85,B 0,C 180,E1 -23931.959,E2 -23931.959} C_VEL
LIN {X 0,Y 151.213,Z 331.619,A -85,B 0,C 180,E1 -23939.999,E2 -23939.999} C_VEL
LIN {X 0,Y 150.681,Z 331.693,A -85,B 0,C 180,E1 -23948.043,E2 -23948.043} C_VEL
LIN {X 0,Y 150.573,Z 331.704,A -85,B 0,C 180,E1 -23951.435,E2 -23951.435} C_VEL
LIN {X 0,Y 150.358,Z 331.753,A -85,B 0,C 180,E1 -23956.287,E2 -23956.287} C_VEL
LIN {X 0,Y 150.346,Z 331.727,A -85,B 0,C 180,E1 -23960.79,E2 -23960.79} C_VEL
LIN {X 0,Y 150.238,Z 331.762,A -85,B 0,C 180,E1 -23967.28,E2 -23967.28} C_VEL
LIN {X 0,Y 150.212,Z 331.762,A -85,B 0,C 180,E1 -23972.633,E2 -23972.633} C_VEL
LIN {X 0,Y 150.169,Z 331.759,A -85,B 0,C 180,E1 -23977.474,E2 -23977.474} C_VEL
LIN {X 0,Y 150.133,Z 331.777,A -85,B 0,C 180,E1 -23981.499,E2 -23981.499} C_VEL
LIN {X 0,Y 150.122,Z 331.766,A -85,B 0,C 180,E1 -23985.396,E2 -23985.396} C_VEL
LIN {X 0,Y 150.148,Z 331.888,A -85,B 0,C 180,E1 -23990.734,E2 -23990.734} C_VEL
LIN {X 0,Y 151.248,Z 334.738,A -85,B 0,C 180,E1 -23991.336,E2 -23991.336} C_VEL
LIN {X 0,Y 153.324,Z 337.228,A -85,B 0,C 180,E1 -23992.25,E2 -23992.25} C_VEL
LIN {X 0,Y 155.65,Z 340.669,A -85,B 0,C 180,E1 -23993.269,E2 -23993.269} C_VEL
LIN {X 0,Y 161.254,Z 349.599,A -85,B 0,C 180,E1 -23995.581,E2 -23995.581} C_VEL
LIN {X 0,Y 166.861,Z 359.492,A -85,B 0,C 180,E1 -23997.727,E2 -23997.727} C_VEL
LIN {X 0,Y 172.98,Z 372.137,A -85,B 0,C 180,E1 -23999.942,E2 -23999.942} C_VEL
LIN {X 0,Y 174.425,Z 375.41,A -85,B 0,C 180,E1 -24000.448,E2 -24000.448} C_VEL
LIN {X 0,Y 171.481,Z 429.85,A -85,B 0,C 180,E1 -24002.549,E2 -24002.549} C_VEL
LIN {X 0,Y 170.206,Z 442.897,A -85,B 0,C 180,E1 -24003.484,E2 -24003.484} C_VEL
LIN {X 0,Y 168.397,Z 455.519,A -85,B 0,C 180,E1 -24004.84,E2 -24004.84} C_VEL
LIN {X 0,Y 165.85,Z 467.628,A -85,B 0,C 180,E1 -24006.593,E2 -24006.593} C_VEL
LIN {X 0,Y 162.79,Z 479.152,A -85,B 0,C 180,E1 -24008.805,E2 -24008.805} C_VEL
LIN {X 0,Y 159.908,Z 489.482,A -85,B 0,C 180,E1 -24011.42,E2 -24011.42} C_VEL
LIN {X 0,Y 156.964,Z 498.786,A -85,B 0,C 180,E1 -24014.417,E2 -24014.417} C_VEL
LIN {X 0,Y 154.041,Z 507.777,A -85,B 0,C 180,E1 -24018.153,E2 -24018.153} C_VEL
LIN {X 0,Y 151.677,Z 515.028,A -85,B 0,C 180,E1 -24022.011,E2 -24022.011} C_VEL
LIN {X 0,Y 149.943,Z 520.832,A -85,B 0,C 180,E1 -24025.969,E2 -24025.969} C_VEL
LIN {X 0,Y 148.707,Z 525.41,A -85,B 0,C 180,E1 -24030.001,E2 -24030.001} C_VEL
LIN {X 0,Y 148.06,Z 529.239,A -85,B 0,C 180,E1 -24034.584,E2 -24034.584} C_VEL
LIN {X 0,Y 147.597,Z 531.403,A -85,B 0,C 180,E1 -24038.214,E2 -24038.214} C_VEL
LIN {X 0,Y 147.538,Z 532.547,A -85,B 0,C 180,E1 -24040.985,E2 -24040.985} C_VEL
LIN {X 0,Y 148.222,Z 533.606,A -85,B 0,C 180,E1 -24046.529,E2 -24046.529} C_VEL
LIN {X 0,Y 148.92,Z 533.553,A -85,B 0,C 180,E1 -24049.291,E2 -24049.291} C_VEL
LIN {X 0,Y 149.796,Z 533.06,A -85,B 0,C 180,E1 -24052.046,E2 -24052.046} C_VEL
LIN {X 0,Y 150.986,Z 532.152,A -85,B 0,C 180,E1 -24054.768,E2 -24054.768} C_VEL
LIN {X 0,Y 152.519,Z 530.84,A -85,B 0,C 180,E1 -24057.439,E2 -24057.439} C_VEL
LIN {X 0,Y 155.213,Z 528.133,A -85,B 0,C 180,E1 -24061.229,E2 -24061.229} C_VEL
LIN {X 0,Y 158.709,Z 524.143,A -85,B 0,C 180,E1 -24065.147,E2 -24065.147} C_VEL
LIN {X 0,Y 163.311,Z 518.319,A -85,B 0,C 180,E1 -24069.23,E2 -24069.23} C_VEL
LIN {X 0,Y 168.244,Z 511.4,A -85,B 0,C 180,E1 -24072.751,E2 -24072.751} C_VEL
LIN {X 0,Y 173.597,Z 503.039,A -85,B 0,C 180,E1 -24075.94,E2 -24075.94} C_VEL
LIN {X 0,Y 178.399,Z 494.399,A -85,B 0,C 180,E1 -24078.461,E2 -24078.461} C_VEL
LIN {X 0,Y 182.914,Z 484.84,A -85,B 0,C 180,E1 -24080.647,E2 -24080.647} C_VEL
LIN {X 0,Y 186.994,Z 474.729,A -85,B 0,C 180,E1 -24082.448,E2 -24082.448} C_VEL
LIN {X 0,Y 190.959,Z 462.844,A -85,B 0,C 180,E1 -24084.065,E2 -24084.065} C_VEL
LIN {X 0,Y 194.002,Z 450.926,A -85,B 0,C 180,E1 -24085.275,E2 -24085.275} C_VEL
LIN {X 0,Y 196.291,Z 438.004,A -85,B 0,C 180,E1 -24086.222,E2 -24086.222} C_VEL
LIN {X 0,Y 197.918,Z 424.949,A -85,B 0,C 180,E1 -24086.755,E2 -24086.755} C_VEL
LIN {X 0,Y 199.783,Z 399.256,A -85,B 0,C 180,E1 -24087.557,E2 -24087.557} C_VEL
LIN {X 0,Y 197.102,Z 393.664,A -85,B 0,C 180,E1 -24088.914,E2 -24088.914} C_VEL
LIN {X 0,Y 191.361,Z 383.469,A -85,B 0,C 180,E1 -24092.005,E2 -24092.005} C_VEL
LIN {X 0,Y 185.042,Z 373.51,A -85,B 0,C 180,E1 -24095.903,E2 -24095.903} C_VEL
LIN {X 0,Y 181.597,Z 368.729,A -85,B 0,C 180,E1 -24098.322,E2 -24098.322} C_VEL
LIN {X 0,Y 178.646,Z 364.615,A -85,B 0,C 180,E1 -24100.656,E2 -24100.656} C_VEL
LIN {X 0,Y 175.972,Z 360.963,A -85,B 0,C 180,E1 -24103.039,E2 -24103.039} C_VEL
LIN {X 0,Y 175.104,Z 359.896,A -85,B 0,C 180,E1 -24103.872,E2 -24103.872} C_VEL
LIN {X 0,Y 172.566,Z 356.627,A -85,B 0,C 180,E1 -24106.607,E2 -24106.607} C_VEL
LIN {X 0,Y 171.836,Z 355.334,A -85,B 0,C 180,E1 -24107.535,E2 -24107.535} C_VEL
LIN {X 0,Y 169.34,Z 352.862,A -85,B 0,C 180,E1 -24110.897,E2 -24110.897} C_VEL
LIN {X 0,Y 167.873,Z 349.908,A -85,B 0,C 180,E1 -24113.691,E2 -24113.691} C_VEL
LIN {X 0,Y 165.247,Z 347.99,A -85,B 0,C 180,E1 -24121.219,E2 -24121.219} C_VEL
LIN {X 0,Y 165.199,Z 348.294,A -85,B 0,C 180,E1 -24128.256,E2 -24128.256} C_VEL
LIN {X 0,Y 167.84,Z 350.192,A -85,B 0,C 180,E1 -24135.847,E2 -24135.847} C_VEL
LIN {X 0,Y 169.367,Z 353.355,A -85,B 0,C 180,E1 -24138.76,E2 -24138.76} C_VEL
LIN {X 0,Y 171.988,Z 355.681,A -85,B 0,C 180,E1 -24142.21,E2 -24142.21} C_VEL
LIN {X 0,Y 174.164,Z 359.083,A -85,B 0,C 180,E1 -24144.751,E2 -24144.751} C_VEL
LIN {X 0,Y 176.608,Z 362.43,A -85,B 0,C 180,E1 -24147.155,E2 -24147.155} C_VEL
LIN {X 0,Y 180.315,Z 368.388,A -85,B 0,C 180,E1 -24150.366,E2 -24150.366} C_VEL
LIN {X 0,Y 183.605,Z 374.181,A -85,B 0,C 180,E1 -24152.876,E2 -24152.876} C_VEL
LIN {X 0,Y 186.833,Z 380.041,A -85,B 0,C 180,E1 -24155.088,E2 -24155.088} C_VEL
LIN {X 0,Y 191.476,Z 389.113,A -85,B 0,C 180,E1 -24157.963,E2 -24157.963} C_VEL
LIN {X 0,Y 196.219,Z 399.874,A -85,B 0,C 180,E1 -24160.65,E2 -24160.65} C_VEL
LIN {X 0,Y 199.339,Z 408.057,A -85,B 0,C 180,E1 -24162.324,E2 -24162.324} C_VEL
LIN {X 0,Y 196.71,Z 440.96,A -85,B 0,C 180,E1 -24163.372,E2 -24163.372} C_VEL
LIN {X 0,Y 194.536,Z 454.495,A -85,B 0,C 180,E1 -24164.108,E2 -24164.108} C_VEL
LIN {X 0,Y 191.559,Z 466.707,A -85,B 0,C 180,E1 -24165.069,E2 -24165.069} C_VEL
LIN {X 0,Y 187.506,Z 479.262,A -85,B 0,C 180,E1 -24166.47,E2 -24166.47} C_VEL
LIN {X 0,Y 183.697,Z 489.161,A -85,B 0,C 180,E1 -24167.969,E2 -24167.969} C_VEL
LIN {X 0,Y 178.917,Z 499.52,A -85,B 0,C 180,E1 -24169.967,E2 -24169.967} C_VEL
LIN {X 0,Y 174.454,Z 508.001,A -85,B 0,C 180,E1 -24172.094,E2 -24172.094} C_VEL
LIN {X 0,Y 169.838,Z 515.843,A -85,B 0,C 180,E1 -24174.596,E2 -24174.596} C_VEL
LIN {X 0,Y 164.722,Z 523.529,A -85,B 0,C 180,E1 -24177.769,E2 -24177.769} C_VEL
LIN {X 0,Y 159.814,Z 530.375,A -85,B 0,C 180,E1 -24181.586,E2 -24181.586} C_VEL
LIN {X 0,Y 156.595,Z 534.668,A -85,B 0,C 180,E1 -24184.762,E2 -24184.762} C_VEL
LIN {X 0,Y 153.954,Z 537.872,A -85,B 0,C 180,E1 -24187.807,E2 -24187.807} C_VEL
LIN {X 0,Y 151.849,Z 539.635,A -85,B 0,C 180,E1 -24189.771,E2 -24189.771} C_VEL
LIN {X 0,Y 147.044,Z 541.884,A -85,B 0,C 180,E1 -24192.98,E2 -24192.98} C_VEL
LIN {X 0,Y 142.696,Z 543.359,A -85,B 0,C 180,E1 -24196.453,E2 -24196.453} C_VEL
LIN {X 0,Y 141.369,Z 543.829,A -85,B 0,C 180,E1 -24198.766,E2 -24198.766} C_VEL
LIN {X 0,Y 140.622,Z 544.126,A -85,B 0,C 180,E1 -24204.262,E2 -24204.262} C_VEL
LIN {X 0,Y 140.636,Z 543.425,A -85,B 0,C 180,E1 -24208.134,E2 -24208.134} C_VEL
LIN {X 0,Y 140.759,Z 542.836,A -85,B 0,C 180,E1 -24209.999,E2 -24209.999} C_VEL
LIN {X 0,Y 140.627,Z 541.558,A -85,B 0,C 180,E1 -24212.864,E2 -24212.864} C_VEL
LIN {X 0,Y 140.763,Z 538.824,A -85,B 0,C 180,E1 -24217.169,E2 -24217.169} C_VEL
LIN {X 0,Y 141.33,Z 535.038,A -85,B 0,C 180,E1 -24221.472,E2 -24221.472} C_VEL
LIN {X 0,Y 142.48,Z 530.102,A -85,B 0,C 180,E1 -24225.74,E2 -24225.74} C_VEL
LIN {X 0,Y 144.503,Z 523.888,A -85,B 0,C 180,E1 -24229.903,E2 -24229.903} C_VEL
LIN {X 0,Y 146.676,Z 517.524,A -85,B 0,C 180,E1 -24233.283,E2 -24233.283} C_VEL
LIN {X 0,Y 149.127,Z 509.854,A -85,B 0,C 180,E1 -24236.594,E2 -24236.594} C_VEL
LIN {X 0,Y 152.194,Z 500.561,A -85,B 0,C 180,E1 -24239.761,E2 -24239.761} C_VEL
LIN {X 0,Y 155.314,Z 490.194,A -85,B 0,C 180,E1 -24242.502,E2 -24242.502} C_VEL
LIN {X 0,Y 158.479,Z 478.702,A -85,B 0,C 180,E1 -24244.816,E2 -24244.816} C_VEL
LIN {X 0,Y 161.258,Z 466.716,A -85,B 0,C 180,E1 -24246.62,E2 -24246.62} C_VEL
LIN {X 0,Y 163.433,Z 454.121,A -85,B 0,C 180,E1 -24247.985,E2 -24247.985} C_VEL
LIN {X 0,Y 164.973,Z 441.127,A -85,B 0,C 180,E1 -24248.928,E2 -24248.928} C_VEL
LIN {X 0,Y 167.655,Z 396.197,A -85,B 0,C 180,E1 -24250.714,E2 -24250.714} C_VEL
LIN {X 0,Y 166.328,Z 379.626,A -85,B 0,C 180,E1 -24251.926,E2 -24251.926} C_VEL
LIN {X 0,Y 160.608,Z 364.304,A -85,B 0,C 180,E1 -24254.361,E2 -24254.361} C_VEL
LIN {X 0,Y 155.153,Z 352.648,A -85,B 0,C 180,E1 -24256.754,E2 -24256.754} C_VEL
LIN {X 0,Y 151.14,Z 345.271,A -85,B 0,C 180,E1 -24258.61,E2 -24258.61} C_VEL
LIN {X 0,Y 148.367,Z 341.272,A -85,B 0,C 180,E1 -24259.914,E2 -24259.914} C_VEL
LIN {X 0,Y 146.099,Z 337.583,A -85,B 0,C 180,E1 -24261.07,E2 -24261.07} C_VEL
LIN {X 0,Y 144.148,Z 335.521,A -85,B 0,C 180,E1 -24262.031,E2 -24262.031} C_VEL
LIN {X 0,Y 143.184,Z 332.986,A -85,B 0,C 180,E1 -24262.633,E2 -24262.633} C_VEL
LIN {X 0,Y 143.143,Z 332.657,A -85,B 0,C 180,E1 -24262.738,E2 -24262.738} C_VEL
LIN {X 0,Y 143.185,Z 332.652,A -85,B 0,C 180,E1 -24267.321,E2 -24267.321} C_VEL
LIN {X 0,Y 143.19,Z 332.649,A -85,B 0,C 180,E1 -24272.06,E2 -24272.06} C_VEL
LIN {X 0,Y 143.275,Z 332.635,A -85,B 0,C 180,E1 -24278.744,E2 -24278.744} C_VEL
LIN {X 0,Y 143.299,Z 332.632,A -85,B 0,C 180,E1 -24282.886,E2 -24282.886} C_VEL
LIN {X 0,Y 143.592,Z 332.566,A -85,B 0,C 180,E1 -24288.709,E2 -24288.709} C_VEL
LIN {X 0,Y 143.659,Z 332.578,A -85,B 0,C 180,E1 -24291.56,E2 -24291.56} C_VEL
LIN {X 0,Y 144.171,Z 332.495,A -85,B 0,C 180,E1 -24299.999,E2 -24299.999} C_VEL
LIN {X 0,Y 143.607,Z 332.569,A -85,B 0,C 180,E1 -24308.442,E2 -24308.442} C_VEL
LIN {X 0,Y 143.501,Z 332.585,A -85,B 0,C 180,E1 -24311.628,E2 -24311.628} C_VEL
LIN {X 0,Y 143.292,Z 332.627,A -85,B 0,C 180,E1 -24317.114,E2 -24317.114} C_VEL
LIN {X 0,Y 143.271,Z 332.609,A -85,B 0,C 180,E1 -24321.252,E2 -24321.252} C_VEL
LIN {X 0,Y 143.185,Z 332.632,A -85,B 0,C 180,E1 -24327.935,E2 -24327.935} C_VEL
LIN {X 0,Y 143.14,Z 332.648,A -85,B 0,C 180,E1 -24333.42,E2 -24333.42} C_VEL
LIN {X 0,Y 143.052,Z 332.642,A -85,B 0,C 180,E1 -24339.693,E2 -24339.693} C_VEL
LIN {X 0,Y 143.048,Z 332.662,A -85,B 0,C 180,E1 -24343.457,E2 -24343.457} C_VEL
LIN {X 0,Y 143.053,Z 332.668,A -85,B 0,C 180,E1 -24347.876,E2 -24347.876} C_VEL
LIN {X 0,Y 143.949,Z 335.284,A -85,B 0,C 180,E1 -24348.457,E2 -24348.457} C_VEL
LIN {X 0,Y 146.086,Z 337.609,A -85,B 0,C 180,E1 -24349.519,E2 -24349.519} C_VEL
LIN {X 0,Y 148.563,Z 341.451,A -85,B 0,C 180,E1 -24350.766,E2 -24350.766} C_VEL
LIN {X 0,Y 154.279,Z 349.896,A -85,B 0,C 180,E1 -24353.376,E2 -24353.376} C_VEL
LIN {X 0,Y 161.094,Z 361.812,A -85,B 0,C 180,E1 -24356.232,E2 -24356.232} C_VEL
LIN {X 0,Y 167.151,Z 374.186,A -85,B 0,C 180,E1 -24358.591,E2 -24358.591} C_VEL
LIN {X 0,Y 168.614,Z 377.809,A -85,B 0,C 180,E1 -24359.158,E2 -24359.158} C_VEL
LIN {X 0,Y 165.608,Z 430.026,A -85,B 0,C 180,E1 -24361.21,E2 -24361.21} C_VEL
LIN {X 0,Y 164.244,Z 443.26,A -85,B 0,C 180,E1 -24362.182,E2 -24362.182} C_VEL
LIN {X 0,Y 162.239,Z 456.414,A -85,B 0,C 180,E1 -24363.641,E2 -24363.641} C_VEL
LIN {X 0,Y 159.786,Z 467.548,A -85,B 0,C 180,E1 -24365.303,E2 -24365.303} C_VEL
LIN {X 0,Y 156.586,Z 479.135,A -85,B 0,C 180,E1 -24367.574,E2 -24367.574} C_VEL
LIN {X 0,Y 153.546,Z 489.515,A -85,B 0,C 180,E1 -24370.273,E2 -24370.273} C_VEL
LIN {X 0,Y 150.735,Z 498.016,A -85,B 0,C 180,E1 -24373.059,E2 -24373.059} C_VEL
LIN {X 0,Y 148.04,Z 505.851,A -85,B 0,C 180,E1 -24376.27,E2 -24376.27} C_VEL
LIN {X 0,Y 145.371,Z 513.502,A -85,B 0,C 180,E1 -24380.259,E2 -24380.259} C_VEL
LIN {X 0,Y 143.395,Z 519.643,A -85,B 0,C 180,E1 -24384.376,E2 -24384.376} C_VEL
LIN {X 0,Y 141.9,Z 524.534,A -85,B 0,C 180,E1 -24388.582,E2 -24388.582} C_VEL
LIN {X 0,Y 141.146,Z 528.3,A -85,B 0,C 180,E1 -24392.855,E2 -24392.855} C_VEL
LIN {X 0,Y 140.763,Z 530.259,A -85,B 0,C 180,E1 -24395.732,E2 -24395.732} C_VEL
LIN {X 0,Y 140.474,Z 531.807,A -85,B 0,C 180,E1 -24398.633,E2 -24398.633} C_VEL
LIN {X 0,Y 140.479,Z 532.895,A -85,B 0,C 180,E1 -24401.545,E2 -24401.545} C_VEL
LIN {X 0,Y 141.281,Z 533.892,A -85,B 0,C 180,E1 -24407.367,E2 -24407.367} C_VEL
LIN {X 0,Y 142.065,Z 533.79,A -85,B 0,C 180,E1 -24410.262,E2 -24410.262} C_VEL
LIN {X 0,Y 144.392,Z 532.31,A -85,B 0,C 180,E1 -24415.981,E2 -24415.981} C_VEL
LIN {X 0,Y 147.816,Z 529.406,A -85,B 0,C 180,E1 -24421.15,E2 -24421.15} C_VEL
LIN {X 0,Y 151.493,Z 525.564,A -85,B 0,C 180,E1 -24425.444,E2 -24425.444} C_VEL
LIN {X 0,Y 155.631,Z 520.816,A -85,B 0,C 180,E1 -24429.214,E2 -24429.214} C_VEL
LIN {X 0,Y 160.398,Z 514.76,A -85,B 0,C 180,E1 -24432.778,E2 -24432.778} C_VEL
LIN {X 0,Y 165.712,Z 507.173,A -85,B 0,C 180,E1 -24436.137,E2 -24436.137} C_VEL
LIN {X 0,Y 170.695,Z 499.233,A -85,B 0,C 180,E1 -24438.795,E2 -24438.795} C_VEL
LIN {X 0,Y 175.768,Z 489.827,A -85,B 0,C 180,E1 -24441.234,E2 -24441.234} C_VEL
LIN {X 0,Y 180.54,Z 479.118,A -85,B 0,C 180,E1 -24443.407,E2 -24443.407} C_VEL
LIN {X 0,Y 184.617,Z 468.422,A -85,B 0,C 180,E1 -24445.034,E2 -24445.034} C_VEL
LIN {X 0,Y 188.182,Z 456.424,A -85,B 0,C 180,E1 -24446.44,E2 -24446.44} C_VEL
LIN {X 0,Y 191.065,Z 443.289,A -85,B 0,C 180,E1 -24447.535,E2 -24447.535} C_VEL
LIN {X 0,Y 192.798,Z 431.886,A -85,B 0,C 180,E1 -24448.169,E2 -24448.169} C_VEL
LIN {X 0,Y 195.175,Z 404.613,A -85,B 0,C 180,E1 -24449.014,E2 -24449.014} C_VEL
LIN {X 0,Y 195.271,Z 401.88,A -85,B 0,C 180,E1 -24449.143,E2 -24449.143} C_VEL
LIN {X 0,Y 190.387,Z 392.512,A -85,B 0,C 180,E1 -24451.84,E2 -24451.84} C_VEL
LIN {X 0,Y 185.724,Z 384.61,A -85,B 0,C 180,E1 -24454.684,E2 -24454.684} C_VEL
LIN {X 0,Y 181.494,Z 377.997,A -85,B 0,C 180,E1 -24457.594,E2 -24457.594} C_VEL
LIN {X 0,Y 179.211,Z 374.666,A -85,B 0,C 180,E1 -24459.333,E2 -24459.333} C_VEL
LIN {X 0,Y 176.535,Z 370.841,A -85,B 0,C 180,E1 -24461.579,E2 -24461.579} C_VEL
LIN {X 0,Y 173.426,Z 366.452,A -85,B 0,C 180,E1 -24464.578,E2 -24464.578} C_VEL
LIN {X 0,Y 170.901,Z 363.044,A -85,B 0,C 180,E1 -24467.466,E2 -24467.466} C_VEL
LIN {X 0,Y 170.202,Z 361.963,A -85,B 0,C 180,E1 -24468.388,E2 -24468.388} C_VEL
LIN {X 0,Y 167.792,Z 359.184,A -85,B 0,C 180,E1 -24471.95,E2 -24471.95} C_VEL
LIN {X 0,Y 166.759,Z 356.876,A -85,B 0,C 180,E1 -24474.104,E2 -24474.104} C_VEL
LIN {X 0,Y 164.373,Z 355.039,A -85,B 0,C 180,E1 -24481.226,E2 -24481.226} C_VEL
LIN {X 0,Y 164.335,Z 355.341,A -85,B 0,C 180,E1 -24488.299,E2 -24488.299} C_VEL
LIN {X 0,Y 166.66,Z 357.12,A -85,B 0,C 180,E1 -24495.305,E2 -24495.305} C_VEL
LIN {X 0,Y 168.229,Z 360.306,A -85,B 0,C 180,E1 -24498.418,E2 -24498.418} C_VEL
LIN {X 0,Y 170.598,Z 362.619,A -85,B 0,C 180,E1 -24501.684,E2 -24501.684} C_VEL
LIN {X 0,Y 174.578,Z 368.551,A -85,B 0,C 180,E1 -24506.184,E2 -24506.184} C_VEL
LIN {X 0,Y 177.996,Z 374.281,A -85,B 0,C 180,E1 -24509.344,E2 -24509.344} C_VEL
LIN {X 0,Y 182.72,Z 382.909,A -85,B 0,C 180,E1 -24513.073,E2 -24513.073} C_VEL
LIN {X 0,Y 187.91,Z 393.432,A -85,B 0,C 180,E1 -24516.597,E2 -24516.597} C_VEL
LIN {X 0,Y 192.58,Z 404.337,A -85,B 0,C 180,E1 -24519.437,E2 -24519.437} C_VEL
LIN {X 0,Y 194.836,Z 410.615,A -85,B 0,C 180,E1 -24520.756,E2 -24520.756} C_VEL
LIN {X 0,Y 192.387,Z 440.385,A -85,B 0,C 180,E1 -24521.715,E2 -24521.715} C_VEL
LIN {X 0,Y 190.172,Z 453.881,A -85,B 0,C 180,E1 -24522.441,E2 -24522.441} C_VEL
LIN {X 0,Y 186.933,Z 466.712,A -85,B 0,C 180,E1 -24523.441,E2 -24523.441} C_VEL
LIN {X 0,Y 183.048,Z 478.418,A -85,B 0,C 180,E1 -24524.74,E2 -24524.74} C_VEL
LIN {X 0,Y 179.629,Z 487.136,A -85,B 0,C 180,E1 -24526.014,E2 -24526.014} C_VEL
LIN {X 0,Y 174.67,Z 497.793,A -85,B 0,C 180,E1 -24528.016,E2 -24528.016} C_VEL
LIN {X 0,Y 168.912,Z 508.287,A -85,B 0,C 180,E1 -24530.615,E2 -24530.615} C_VEL
LIN {X 0,Y 163.169,Z 517.382,A -85,B 0,C 180,E1 -24533.683,E2 -24533.683} C_VEL
LIN {X 0,Y 157.928,Z 524.733,A -85,B 0,C 180,E1 -24536.965,E2 -24536.965} C_VEL
LIN {X 0,Y 153.23,Z 530.856,A -85,B 0,C 180,E1 -24540.629,E2 -24540.629} C_VEL
LIN {X 0,Y 148.952,Z 536.024,A -85,B 0,C 180,E1 -24544.871,E2 -24544.871} C_VEL
LIN {X 0,Y 146.819,Z 538.413,A -85,B 0,C 180,E1 -24547.483,E2 -24547.483} C_VEL
LIN {X 0,Y 143.356,Z 541.942,A -85,B 0,C 180,E1 -24552.893,E2 -24552.893} C_VEL
LIN {X 0,Y 141.425,Z 543.8,A -85,B 0,C 180,E1 -24558.534,E2 -24558.534} C_VEL
LIN {X 0,Y 141.369,Z 543.829,A -85,B 0,C 180,E1 -24558.766,E2 -24558.766} C_VEL
LIN {X 0,Y 140.296,Z 544.134,A -85,B 0,C 180,E1 -24561.131,E2 -24561.131} C_VEL
LIN {X 0,Y 137.216,Z 543.88,A -85,B 0,C 180,E1 -24565.023,E2 -24565.023} C_VEL
LIN {X 0,Y 134.782,Z 543.179,A -85,B 0,C 180,E1 -24568.227,E2 -24568.227} C_VEL
LIN {X 0,Y 133.577,Z 541.884,A -85,B 0,C 180,E1 -24571.549,E2 -24571.549} C_VEL
LIN {X 0,Y 133.622,Z 539.457,A -85,B 0,C 180,E1 -24576.037,E2 -24576.037} C_VEL
LIN {X 0,Y 134.069,Z 535.974,A -85,B 0,C 180,E1 -24580.571,E2 -24580.571} C_VEL
LIN {X 0,Y 135.119,Z 531.376,A -85,B 0,C 180,E1 -24585.073,E2 -24585.073} C_VEL
LIN {X 0,Y 137.385,Z 524.396,A -85,B 0,C 180,E1 -24590.199,E2 -24590.199} C_VEL
LIN {X 0,Y 140.156,Z 516.839,A -85,B 0,C 180,E1 -24594.43,E2 -24594.43} C_VEL
LIN {X 0,Y 142.324,Z 510.261,A -85,B 0,C 180,E1 -24597.396,E2 -24597.396} C_VEL
LIN {X 0,Y 145.683,Z 500.669,A -85,B 0,C 180,E1 -24600.834,E2 -24600.834} C_VEL
LIN {X 0,Y 148.948,Z 490.413,A -85,B 0,C 180,E1 -24603.669,E2 -24603.669} C_VEL
LIN {X 0,Y 152.249,Z 479.029,A -85,B 0,C 180,E1 -24606.053,E2 -24606.053} C_VEL
LIN {X 0,Y 155.133,Z 467.211,A -85,B 0,C 180,E1 -24607.908,E2 -24607.908} C_VEL
LIN {X 0,Y 157.472,Z 454.422,A -85,B 0,C 180,E1 -24609.36,E2 -24609.36} C_VEL
LIN {X 0,Y 159.134,Z 441.219,A -85,B 0,C 180,E1 -24610.352,E2 -24610.352} C_VEL
LIN {X 0,Y 161.42,Z 406.568,A -85,B 0,C 180,E1 -24611.765,E2 -24611.765} C_VEL
LIN {X 0,Y 161.865,Z 395.493,A -85,B 0,C 180,E1 -24612.255,E2 -24612.255} C_VEL
LIN {X 0,Y 160.821,Z 382.113,A -85,B 0,C 180,E1 -24613.289,E2 -24613.289} C_VEL
LIN {X 0,Y 155.521,Z 367.596,A -85,B 0,C 180,E1 -24615.727,E2 -24615.727} C_VEL
LIN {X 0,Y 150.149,Z 355.968,A -85,B 0,C 180,E1 -24618.276,E2 -24618.276} C_VEL
LIN {X 0,Y 146.922,Z 349.98,A -85,B 0,C 180,E1 -24619.885,E2 -24619.885} C_VEL
LIN {X 0,Y 141.978,Z 342.729,A -85,B 0,C 180,E1 -24622.448,E2 -24622.448} C_VEL
LIN {X 0,Y 139.793,Z 339.522,A -85,B 0,C 180,E1 -24623.679,E2 -24623.679} C_VEL
LIN {X 0,Y 139.162,Z 338.585,A -85,B 0,C 180,E1 -24624.048,E2 -24624.048} C_VEL
LIN {X 0,Y 137.044,Z 336.386,A -85,B 0,C 180,E1 -24625.258,E2 -24625.258} C_VEL
LIN {X 0,Y 136.135,Z 333.91,A -85,B 0,C 180,E1 -24625.925,E2 -24625.925} C_VEL
LIN {X 0,Y 136.1,Z 333.535,A -85,B 0,C 180,E1 -24626.063,E2 -24626.063} C_VEL
LIN {X 0,Y 136.146,Z 333.528,A -85,B 0,C 180,E1 -24632.316,E2 -24632.316} C_VEL
LIN {X 0,Y 136.242,Z 333.511,A -85,B 0,C 180,E1 -24638.832,E2 -24638.832} C_VEL
LIN {X 0,Y 136.269,Z 333.507,A -85,B 0,C 180,E1 -24645.056,E2 -24645.056} C_VEL
LIN {X 0,Y 136.495,Z 333.451,A -85,B 0,C 180,E1 -24648.114,E2 -24648.114} C_VEL
LIN {X 0,Y 136.586,Z 333.451,A -85,B 0,C 180,E1 -24651.119,E2 -24651.119} C_VEL
LIN {X 0,Y 137.128,Z 333.371,A -85,B 0,C 180,E1 -24659.999,E2 -24659.999} C_VEL
LIN {X 0,Y 136.536,Z 333.445,A -85,B 0,C 180,E1 -24668.883,E2 -24668.883} C_VEL
LIN {X 0,Y 136.437,Z 333.466,A -85,B 0,C 180,E1 -24671.89,E2 -24671.89} C_VEL
LIN {X 0,Y 136.206,Z 333.499,A -85,B 0,C 180,E1 -24678.034,E2 -24678.034} C_VEL
LIN {X 0,Y 136.192,Z 333.492,A -85,B 0,C 180,E1 -24681.746,E2 -24681.746} C_VEL
LIN {X 0,Y 136.095,Z 333.507,A -85,B 0,C 180,E1 -24688.615,E2 -24688.615} C_VEL
LIN {X 0,Y 136.04,Z 333.538,A -85,B 0,C 180,E1 -24694.629,E2 -24694.629} C_VEL
LIN {X 0,Y 136.024,Z 333.515,A -85,B 0,C 180,E1 -24699.196,E2 -24699.196} C_VEL
LIN {X 0,Y 135.957,Z 333.534,A -85,B 0,C 180,E1 -24704.514,E2 -24704.514} C_VEL
LIN {X 0,Y 136.859,Z 336.239,A -85,B 0,C 180,E1 -24705.23,E2 -24705.23} C_VEL
LIN {X 0,Y 138.752,Z 338.326,A -85,B 0,C 180,E1 -24706.328,E2 -24706.328} C_VEL
LIN {X 0,Y 139.542,Z 339.061,A -85,B 0,C 180,E1 -24706.76,E2 -24706.76} C_VEL
LIN {X 0,Y 141.646,Z 342.393,A -85,B 0,C 180,E1 -24707.972,E2 -24707.972} C_VEL
LIN {X 0,Y 143.031,Z 344.18,A -85,B 0,C 180,E1 -24708.707,E2 -24708.707} C_VEL
LIN {X 0,Y 148.523,Z 352.335,A -85,B 0,C 180,E1 -24711.479,E2 -24711.479} C_VEL
LIN {X 0,Y 153.838,Z 361.22,A -85,B 0,C 180,E1 -24713.929,E2 -24713.929} C_VEL
LIN {X 0,Y 160.355,Z 374.048,A -85,B 0,C 180,E1 -24716.712,E2 -24716.712} C_VEL
LIN {X 0,Y 162.714,Z 379.404,A -85,B 0,C 180,E1 -24717.682,E2 -24717.682} C_VEL
LIN {X 0,Y 162.207,Z 391.084,A -85,B 0,C 180,E1 -24718.188,E2 -24718.188} C_VEL
LIN {X 0,Y 159.744,Z 431.087,A -85,B 0,C 180,E1 -24719.827,E2 -24719.827} C_VEL
LIN {X 0,Y 158.183,Z 445.127,A -85,B 0,C 180,E1 -24720.927,E2 -24720.927} C_VEL
LIN {X 0,Y 156.166,Z 457.265,A -85,B 0,C 180,E1 -24722.35,E2 -24722.35} C_VEL
LIN {X 0,Y 153.36,Z 469.055,A -85,B 0,C 180,E1 -24724.193,E2 -24724.193} C_VEL
LIN {X 0,Y 150.101,Z 480.402,A -85,B 0,C 180,E1 -24726.549,E2 -24726.549} C_VEL
LIN {X 0,Y 146.906,Z 490.601,A -85,B 0,C 180,E1 -24729.341,E2 -24729.341} C_VEL
LIN {X 0,Y 143.373,Z 500.586,A -85,B 0,C 180,E1 -24732.897,E2 -24732.897} C_VEL
LIN {X 0,Y 140.222,Z 509.362,A -85,B 0,C 180,E1 -24736.966,E2 -24736.966} C_VEL
LIN {X 0,Y 137.658,Z 516.392,A -85,B 0,C 180,E1 -24741.191,E2 -24741.191} C_VEL
LIN {X 0,Y 135.773,Z 522.006,A -85,B 0,C 180,E1 -24745.548,E2 -24745.548} C_VEL
LIN {X 0,Y 134.526,Z 526.431,A -85,B 0,C 180,E1 -24750.001,E2 -24750.001} C_VEL
LIN {X 0,Y 133.908,Z 529.661,A -85,B 0,C 180,E1 -24754.302,E2 -24754.302} C_VEL
LIN {X 0,Y 133.38,Z 532.189,A -85,B 0,C 180,E1 -24759.096,E2 -24759.096} C_VEL
LIN {X 0,Y 133.425,Z 533.242,A -85,B 0,C 180,E1 -24762.164,E2 -24762.164} C_VEL
LIN {X 0,Y 134.38,Z 534.177,A -85,B 0,C 180,E1 -24768.289,E2 -24768.289} C_VEL
LIN {X 0,Y 135.238,Z 534.014,A -85,B 0,C 180,E1 -24771.333,E2 -24771.333} C_VEL
LIN {X 0,Y 137.871,Z 532.468,A -85,B 0,C 180,E1 -24777.309,E2 -24777.309} C_VEL
LIN {X 0,Y 141.251,Z 529.792,A -85,B 0,C 180,E1 -24782.239,E2 -24782.239} C_VEL
LIN {X 0,Y 145.594,Z 525.548,A -85,B 0,C 180,E1 -24787.114,E2 -24787.114} C_VEL
LIN {X 0,Y 150.027,Z 520.724,A -85,B 0,C 180,E1 -24790.983,E2 -24790.983} C_VEL
LIN {X 0,Y 155.123,Z 514.585,A -85,B 0,C 180,E1 -24794.608,E2 -24794.608} C_VEL
LIN {X 0,Y 160.757,Z 506.903,A -85,B 0,C 180,E1 -24798.006,E2 -24798.006} C_VEL
LIN {X 0,Y 166.164,Z 498.487,A -85,B 0,C 180,E1 -24800.787,E2 -24800.787} C_VEL
LIN {X 0,Y 171.829,Z 488.158,A -85,B 0,C 180,E1 -24803.388,E2 -24803.388} C_VEL
LIN {X 0,Y 176.297,Z 478.367,A -85,B 0,C 180,E1 -24805.307,E2 -24805.307} C_VEL
LIN {X 0,Y 180.568,Z 467.409,A -85,B 0,C 180,E1 -24806.916,E2 -24806.916} C_VEL
LIN {X 0,Y 184.246,Z 454.994,A -85,B 0,C 180,E1 -24808.314,E2 -24808.314} C_VEL
LIN {X 0,Y 187.03,Z 442.338,A -85,B 0,C 180,E1 -24809.332,E2 -24809.332} C_VEL
LIN {X 0,Y 188.873,Z 429.928,A -85,B 0,C 180,E1 -24809.974,E2 -24809.974} C_VEL
LIN {X 0,Y 190.961,Z 404.931,A -85,B 0,C 180,E1 -24810.758,E2 -24810.758} C_VEL
LIN {X 0,Y 186.404,Z 396.246,A -85,B 0,C 180,E1 -24813.478,E2 -24813.478} C_VEL
LIN {X 0,Y 182.06,Z 388.582,A -85,B 0,C 180,E1 -24816.386,E2 -24816.386} C_VEL
LIN {X 0,Y 177.482,Z 381.403,A -85,B 0,C 180,E1 -24819.879,E2 -24819.879} C_VEL
LIN {X 0,Y 174.395,Z 376.949,A -85,B 0,C 180,E1 -24822.597,E2 -24822.597} C_VEL
LIN {X 0,Y 171.736,Z 373.002,A -85,B 0,C 180,E1 -24825.333,E2 -24825.333} C_VEL
LIN {X 0,Y 169.238,Z 369.369,A -85,B 0,C 180,E1 -24828.396,E2 -24828.396} C_VEL
LIN {X 0,Y 168.258,Z 368.272,A -85,B 0,C 180,E1 -24829.737,E2 -24829.737} C_VEL
LIN {X 0,Y 166.027,Z 364.856,A -85,B 0,C 180,E1 -24833.621,E2 -24833.621} C_VEL
LIN {X 0,Y 165.654,Z 363.84,A -85,B 0,C 180,E1 -24834.523,E2 -24834.523} C_VEL
LIN {X 0,Y 163.5,Z 362.087,A -85,B 0,C 180,E1 -24841.232,E2 -24841.232} C_VEL
LIN {X 0,Y 163.53,Z 362.48,A -85,B 0,C 180,E1 -24848.707,E2 -24848.707} C_VEL
LIN {X 0,Y 165.502,Z 364.013,A -85,B 0,C 180,E1 -24854.762,E2 -24854.762} C_VEL
LIN {X 0,Y 167.097,Z 367.259,A -85,B 0,C 180,E1 -24858.071,E2 -24858.071} C_VEL
LIN {X 0,Y 169.173,Z 369.443,A -85,B 0,C 180,E1 -24861.077,E2 -24861.077} C_VEL
LIN {X 0,Y 172.694,Z 374.893,A -85,B 0,C 180,E1 -24865.298,E2 -24865.298} C_VEL
LIN {X 0,Y 175.929,Z 380.609,A -85,B 0,C 180,E1 -24868.482,E2 -24868.482} C_VEL
LIN {X 0,Y 180.036,Z 388.461,A -85,B 0,C 180,E1 -24871.942,E2 -24871.942} C_VEL
LIN {X 0,Y 184.56,Z 398.024,A -85,B 0,C 180,E1 -24875.251,E2 -24875.251} C_VEL
LIN {X 0,Y 188.746,Z 408.011,A -85,B 0,C 180,E1 -24877.995,E2 -24877.995} C_VEL
LIN {X 0,Y 190.462,Z 412.81,A -85,B 0,C 180,E1 -24879.076,E2 -24879.076} C_VEL
LIN {X 0,Y 188.23,Z 439.809,A -85,B 0,C 180,E1 -24879.978,E2 -24879.978} C_VEL
LIN {X 0,Y 185.927,Z 453.399,A -85,B 0,C 180,E1 -24880.692,E2 -24880.692} C_VEL
LIN {X 0,Y 182.787,Z 465.718,A -85,B 0,C 180,E1 -24881.638,E2 -24881.638} C_VEL
LIN {X 0,Y 178.757,Z 477.594,A -85,B 0,C 180,E1 -24882.923,E2 -24882.923} C_VEL
LIN {X 0,Y 174.615,Z 487.701,A -85,B 0,C 180,E1 -24884.404,E2 -24884.404} C_VEL
LIN {X 0,Y 169.481,Z 498.214,A -85,B 0,C 180,E1 -24886.417,E2 -24886.417} C_VEL
LIN {X 0,Y 164.57,Z 506.824,A -85,B 0,C 180,E1 -24888.552,E2 -24888.552} C_VEL
LIN {X 0,Y 159.47,Z 514.771,A -85,B 0,C 180,E1 -24891.096,E2 -24891.096} C_VEL
LIN {X 0,Y 153.774,Z 522.586,A -85,B 0,C 180,E1 -24894.357,E2 -24894.357} C_VEL
LIN {X 0,Y 149.507,Z 527.909,A -85,B 0,C 180,E1 -24897.275,E2 -24897.275} C_VEL
LIN {X 0,Y 145.177,Z 533.129,A -85,B 0,C 180,E1 -24901.046,E2 -24901.046} C_VEL
LIN {X 0,Y 141.343,Z 537.207,A -85,B 0,C 180,E1 -24904.997,E2 -24904.997} C_VEL
LIN {X 0,Y 138.238,Z 540.255,A -85,B 0,C 180,E1 -24909.152,E2 -24909.152} C_VEL
LIN {X 0,Y 136.554,Z 541.777,A -85,B 0,C 180,E1 -24912.012,E2 -24912.012} C_VEL
LIN {X 0,Y 134.458,Z 543.572,A -85,B 0,C 180,E1 -24917.931,E2 -24917.931} C_VEL
LIN {X 0,Y 133.549,Z 543.845,A -85,B 0,C 180,E1 -24923.957,E2 -24923.957} C_VEL
LIN {X 0,Y 133.571,Z 542.944,A -85,B 0,C 180,E1 -24928.642,E2 -24928.642} C_VEL
LIN {X 0,Y 133.577,Z 541.884,A -85,B 0,C 180,E1 -24931.549,E2 -24931.549} C_VEL
LIN {X 0,Y 132.835,Z 540.64,A -85,B 0,C 180,E1 -24934.008,E2 -24934.008} C_VEL
LIN {X 0,Y 130.168,Z 537.992,A -85,B 0,C 180,E1 -24938.017,E2 -24938.017} C_VEL
LIN {X 0,Y 128.197,Z 535.405,A -85,B 0,C 180,E1 -24941.262,E2 -24941.262} C_VEL
LIN {X 0,Y 127.681,Z 533.127,A -85,B 0,C 180,E1 -24943.718,E2 -24943.718} C_VEL
LIN {X 0,Y 127.807,Z 532.289,A -85,B 0,C 180,E1 -24944.526,E2 -24944.526} C_VEL
LIN {X 0,Y 129.895,Z 525.999,A -85,B 0,C 180,E1 -24949.763,E2 -24949.763} C_VEL
LIN {X 0,Y 132.544,Z 518.867,A -85,B 0,C 180,E1 -24954.262,E2 -24954.262} C_VEL
LIN {X 0,Y 135.186,Z 511.572,A -85,B 0,C 180,E1 -24957.896,E2 -24957.896} C_VEL
LIN {X 0,Y 138.452,Z 502.735,A -85,B 0,C 180,E1 -24961.351,E2 -24961.351} C_VEL
LIN {X 0,Y 142.199,Z 491.847,A -85,B 0,C 180,E1 -24964.635,E2 -24964.635} C_VEL
LIN {X 0,Y 145.646,Z 480.951,A -85,B 0,C 180,E1 -24967.096,E2 -24967.096} C_VEL
LIN {X 0,Y 148.831,Z 468.683,A -85,B 0,C 180,E1 -24969.166,E2 -24969.166} C_VEL
LIN {X 0,Y 151.423,Z 456.019,A -85,B 0,C 180,E1 -24970.709,E2 -24970.709} C_VEL
LIN {X 0,Y 153.269,Z 442.937,A -85,B 0,C 180,E1 -24971.773,E2 -24971.773} C_VEL
LIN {X 0,Y 154.647,Z 424.426,A -85,B 0,C 180,E1 -24972.639,E2 -24972.639} C_VEL
LIN {X 0,Y 156.298,Z 396.841,A -85,B 0,C 180,E1 -24973.758,E2 -24973.758} C_VEL
LIN {X 0,Y 155.402,Z 384.388,A -85,B 0,C 180,E1 -24974.761,E2 -24974.761} C_VEL
LIN {X 0,Y 150.284,Z 370.313,A -85,B 0,C 180,E1 -24977.305,E2 -24977.305} C_VEL
LIN {X 0,Y 145.179,Z 359.02,A -85,B 0,C 180,E1 -24979.95,E2 -24979.95} C_VEL
LIN {X 0,Y 142.027,Z 353.454,A -85,B 0,C 180,E1 -24981.643,E2 -24981.643} C_VEL
LIN {X 0,Y 138.035,Z 347.685,A -85,B 0,C 180,E1 -24983.878,E2 -24983.878} C_VEL
LIN {X 0,Y 135.647,Z 344.21,A -85,B 0,C 180,E1 -24985.331,E2 -24985.331} C_VEL
LIN {X 0,Y 133.246,Z 341.068,A -85,B 0,C 180,E1 -24986.863,E2 -24986.863} C_VEL
LIN {X 0,Y 132.496,Z 339.627,A -85,B 0,C 180,E1 -24987.404,E2 -24987.404} C_VEL
LIN {X 0,Y 130.317,Z 337.703,A -85,B 0,C 180,E1 -24988.843,E2 -24988.843} C_VEL
LIN {X 0,Y 129.199,Z 335.288,A -85,B 0,C 180,E1 -24989.756,E2 -24989.756} C_VEL
LIN {X 0,Y 129.032,Z 334.417,A -85,B 0,C 180,E1 -24990.04,E2 -24990.04} C_VEL
LIN {X 0,Y 129.029,Z 334.412,A -85,B 0,C 180,E1 -24994.166,E2 -24994.166} C_VEL
LIN {X 0,Y 129.106,Z 334.401,A -85,B 0,C 180,E1 -24997.727,E2 -24997.727} C_VEL
LIN {X 0,Y 129.151,Z 334.396,A -85,B 0,C 180,E1 -25000.943,E2 -25000.943} C_VEL
LIN {X 0,Y 129.414,Z 334.333,A -85,B 0,C 180,E1 -25007.819,E2 -25007.819} C_VEL
LIN {X 0,Y 129.513,Z 334.326,A -85,B 0,C 180,E1 -25010.63,E2 -25010.63} C_VEL
LIN {X 0,Y 130.084,Z 334.247,A -85,B 0,C 180,E1 -25019.999,E2 -25019.999} C_VEL
LIN {X 0,Y 129.462,Z 334.323,A -85,B 0,C 180,E1 -25029.372,E2 -25029.372} C_VEL
LIN {X 0,Y 129.341,Z 334.356,A -85,B 0,C 180,E1 -25032.553,E2 -25032.553} C_VEL
LIN {X 0,Y 129.127,Z 334.37,A -85,B 0,C 180,E1 -25039.06,E2 -25039.06} C_VEL
LIN {X 0,Y 129.104,Z 334.379,A -85,B 0,C 180,E1 -25042.398,E2 -25042.398} C_VEL
LIN {X 0,Y 129.024,Z 334.413,A -85,B 0,C 180,E1 -25045.833,E2 -25045.833} C_VEL
LIN {X 0,Y 129.013,Z 334.384,A -85,B 0,C 180,E1 -25049.358,E2 -25049.358} C_VEL
LIN {X 0,Y 128.956,Z 334.419,A -85,B 0,C 180,E1 -25055.168,E2 -25055.168} C_VEL
LIN {X 0,Y 128.936,Z 334.404,A -85,B 0,C 180,E1 -25060.532,E2 -25060.532} C_VEL
LIN {X 0,Y 129.839,Z 337.08,A -85,B 0,C 180,E1 -25061.405,E2 -25061.405} C_VEL
LIN {X 0,Y 131.864,Z 339.315,A -85,B 0,C 180,E1 -25062.807,E2 -25062.807} C_VEL
LIN {X 0,Y 132.642,Z 339.942,A -85,B 0,C 180,E1 -25063.302,E2 -25063.302} C_VEL
LIN {X 0,Y 134.485,Z 343.065,A -85,B 0,C 180,E1 -25064.569,E2 -25064.569} C_VEL
LIN {X 0,Y 136.309,Z 345.126,A -85,B 0,C 180,E1 -25065.674,E2 -25065.674} C_VEL
LIN {X 0,Y 140.22,Z 350.865,A -85,B 0,C 180,E1 -25067.97,E2 -25067.97} C_VEL
LIN {X 0,Y 144.946,Z 357.981,A -85,B 0,C 180,E1 -25070.477,E2 -25070.477} C_VEL
LIN {X 0,Y 150.927,Z 368.553,A -85,B 0,C 180,E1 -25073.399,E2 -25073.399} C_VEL
LIN {X 0,Y 156.495,Z 380.107,A -85,B 0,C 180,E1 -25075.915,E2 -25075.915} C_VEL
LIN {X 0,Y 157.14,Z 381.684,A -85,B 0,C 180,E1 -25076.203,E2 -25076.203} C_VEL
LIN {X 0,Y 154.077,Z 431.088,A -85,B 0,C 180,E1 -25078.273,E2 -25078.273} C_VEL
LIN {X 0,Y 152.516,Z 444.698,A -85,B 0,C 180,E1 -25079.35,E2 -25079.35} C_VEL
LIN {X 0,Y 150.393,Z 457.074,A -85,B 0,C 180,E1 -25080.808,E2 -25080.808} C_VEL
LIN {X 0,Y 147.464,Z 468.971,A -85,B 0,C 180,E1 -25082.697,E2 -25082.697} C_VEL
LIN {X 0,Y 144.045,Z 480.383,A -85,B 0,C 180,E1 -25085.115,E2 -25085.115} C_VEL
LIN {X 0,Y 140.666,Z 490.642,A -85,B 0,C 180,E1 -25087.994,E2 -25087.994} C_VEL
LIN {X 0,Y 137.256,Z 499.86,A -85,B 0,C 180,E1 -25091.337,E2 -25091.337} C_VEL
LIN {X 0,Y 133.842,Z 508.803,A -85,B 0,C 180,E1 -25095.558,E2 -25095.558} C_VEL
LIN {X 0,Y 131.051,Z 516.014,A -85,B 0,C 180,E1 -25099.964,E2 -25099.964} C_VEL
LIN {X 0,Y 129.305,Z 520.878,A -85,B 0,C 180,E1 -25103.761,E2 -25103.761} C_VEL
LIN {X 0,Y 127.714,Z 525.621,A -85,B 0,C 180,E1 -25108.424,E2 -25108.424} C_VEL
LIN {X 0,Y 126.907,Z 529.25,A -85,B 0,C 180,E1 -25113.176,E2 -25113.176} C_VEL
LIN {X 0,Y 126.47,Z 531.143,A -85,B 0,C 180,E1 -25116.382,E2 -25116.382} C_VEL
LIN {X 0,Y 126.277,Z 532.569,A -85,B 0,C 180,E1 -25119.613,E2 -25119.613} C_VEL
LIN {X 0,Y 126.778,Z 534.222,A -85,B 0,C 180,E1 -25126.093,E2 -25126.093} C_VEL
LIN {X 0,Y 128.009,Z 534.378,A -85,B 0,C 180,E1 -25131.041,E2 -25131.041} C_VEL
LIN {X 0,Y 129.793,Z 533.631,A -85,B 0,C 180,E1 -25135.671,E2 -25135.671} C_VEL
LIN {X 0,Y 131.434,Z 532.627,A -85,B 0,C 180,E1 -25138.768,E2 -25138.768} C_VEL
LIN {X 0,Y 134.759,Z 530.164,A -85,B 0,C 180,E1 -25143.444,E2 -25143.444} C_VEL
LIN {X 0,Y 138.421,Z 526.917,A -85,B 0,C 180,E1 -25147.538,E2 -25147.538} C_VEL
LIN {X 0,Y 142.956,Z 522.427,A -85,B 0,C 180,E1 -25151.582,E2 -25151.582} C_VEL
LIN {X 0,Y 148.148,Z 516.672,A -85,B 0,C 180,E1 -25155.365,E2 -25155.365} C_VEL
LIN {X 0,Y 153.919,Z 509.39,A -85,B 0,C 180,E1 -25158.886,E2 -25158.886} C_VEL
LIN {X 0,Y 160.326,Z 500.22,A -85,B 0,C 180,E1 -25162.143,E2 -25162.143} C_VEL
LIN {X 0,Y 165.898,Z 490.856,A -85,B 0,C 180,E1 -25164.637,E2 -25164.637} C_VEL
LIN {X 0,Y 171.066,Z 480.251,A -85,B 0,C 180,E1 -25166.834,E2 -25166.834} C_VEL
LIN {X 0,Y 175.582,Z 469.383,A -85,B 0,C 180,E1 -25168.498,E2 -25168.498} C_VEL
LIN {X 0,Y 179.515,Z 457.235,A -85,B 0,C 180,E1 -25169.929,E2 -25169.929} C_VEL
LIN {X 0,Y 182.637,Z 444.115,A -85,B 0,C 180,E1 -25171.02,E2 -25171.02} C_VEL
LIN {X 0,Y 184.66,Z 431.771,A -85,B 0,C 180,E1 -25171.69,E2 -25171.69} C_VEL
LIN {X 0,Y 186.799,Z 408.092,A -85,B 0,C 180,E1 -25172.443,E2 -25172.443} C_VEL
LIN {X 0,Y 181.528,Z 397.925,A -85,B 0,C 180,E1 -25175.938,E2 -25175.938} C_VEL
LIN {X 0,Y 176.939,Z 390.155,A -85,B 0,C 180,E1 -25179.435,E2 -25179.435} C_VEL
LIN {X 0,Y 172.954,Z 383.842,A -85,B 0,C 180,E1 -25183.019,E2 -25183.019} C_VEL
LIN {X 0,Y 170.078,Z 379.549,A -85,B 0,C 180,E1 -25186.103,E2 -25186.103} C_VEL
LIN {X 0,Y 167.25,Z 375.333,A -85,B 0,C 180,E1 -25189.866,E2 -25189.866} C_VEL
LIN {X 0,Y 165.055,Z 372.199,A -85,B 0,C 180,E1 -25193.698,E2 -25193.698} C_VEL
LIN {X 0,Y 164.489,Z 370.757,A -85,B 0,C 180,E1 -25195.098,E2 -25195.098} C_VEL
LIN {X 0,Y 162.628,Z 369.124,A -85,B 0,C 180,E1 -25201.239,E2 -25201.239} C_VEL
LIN {X 0,Y 162.654,Z 369.545,A -85,B 0,C 180,E1 -25208.702,E2 -25208.702} C_VEL
LIN {X 0,Y 164.413,Z 371.063,A -85,B 0,C 180,E1 -25214.36,E2 -25214.36} C_VEL
LIN {X 0,Y 165.971,Z 374.217,A -85,B 0,C 180,E1 -25217.72,E2 -25217.72} C_VEL
LIN {X 0,Y 167.722,Z 376.144,A -85,B 0,C 180,E1 -25220.385,E2 -25220.385} C_VEL
LIN {X 0,Y 170.782,Z 381.036,A -85,B 0,C 180,E1 -25224.301,E2 -25224.301} C_VEL
LIN {X 0,Y 173.858,Z 386.811,A -85,B 0,C 180,E1 -25227.553,E2 -25227.553} C_VEL
LIN {X 0,Y 177.564,Z 394.288,A -85,B 0,C 180,E1 -25230.892,E2 -25230.892} C_VEL
LIN {X 0,Y 181.591,Z 403.198,A -85,B 0,C 180,E1 -25234.055,E2 -25234.055} C_VEL
LIN {X 0,Y 185.443,Z 412.968,A -85,B 0,C 180,E1 -25236.785,E2 -25236.785} C_VEL
LIN {X 0,Y 186.302,Z 415.448,A -85,B 0,C 180,E1 -25237.371,E2 -25237.371} C_VEL
LIN {X 0,Y 184.106,Z 440.321,A -85,B 0,C 180,E1 -25238.213,E2 -25238.213} C_VEL
LIN {X 0,Y 181.788,Z 453.314,A -85,B 0,C 180,E1 -25238.893,E2 -25238.893} C_VEL
LIN {X 0,Y 178.502,Z 465.758,A -85,B 0,C 180,E1 -25239.847,E2 -25239.847} C_VEL
LIN {X 0,Y 174.03,Z 478.345,A -85,B 0,C 180,E1 -25241.222,E2 -25241.222} C_VEL
LIN {X 0,Y 170.295,Z 486.987,A -85,B 0,C 180,E1 -25242.464,E2 -25242.464} C_VEL
LIN {X 0,Y 165.006,Z 497.571,A -85,B 0,C 180,E1 -25244.485,E2 -25244.485} C_VEL
LIN {X 0,Y 159.329,Z 507.132,A -85,B 0,C 180,E1 -25246.865,E2 -25246.865} C_VEL
LIN {X 0,Y 154.006,Z 514.985,A -85,B 0,C 180,E1 -25249.436,E2 -25249.436} C_VEL
LIN {X 0,Y 148.062,Z 522.682,A -85,B 0,C 180,E1 -25252.756,E2 -25252.756} C_VEL
LIN {X 0,Y 141.953,Z 529.789,A -85,B 0,C 180,E1 -25257.002,E2 -25257.002} C_VEL
LIN {X 0,Y 137.585,Z 534.549,A -85,B 0,C 180,E1 -25260.969,E2 -25260.969} C_VEL
LIN {X 0,Y 133.738,Z 538.219,A -85,B 0,C 180,E1 -25265.139,E2 -25265.139} C_VEL
LIN {X 0,Y 131.601,Z 540.132,A -85,B 0,C 180,E1 -25268.047,E2 -25268.047} C_VEL
LIN {X 0,Y 129.788,Z 541.602,A -85,B 0,C 180,E1 -25271.04,E2 -25271.04} C_VEL
LIN {X 0,Y 127.486,Z 543.344,A -85,B 0,C 180,E1 -25277.26,E2 -25277.26} C_VEL
LIN {X 0,Y 126.852,Z 543.648,A -85,B 0,C 180,E1 -25280.431,E2 -25280.431} C_VEL
LIN {X 0,Y 126.471,Z 543.552,A -85,B 0,C 180,E1 -25283.618,E2 -25283.618} C_VEL
LIN {X 0,Y 126.516,Z 542.375,A -85,B 0,C 180,E1 -25289.283,E2 -25289.283} C_VEL
LIN {X 0,Y 126.45,Z 540.8,A -85,B 0,C 180,E1 -25293.185,E2 -25293.185} C_VEL
LIN {X 0,Y 126.648,Z 537.956,A -85,B 0,C 180,E1 -25297.973,E2 -25297.973} C_VEL
LIN {X 0,Y 127.36,Z 534.053,A -85,B 0,C 180,E1 -25302.751,E2 -25302.751} C_VEL
LIN {X 0,Y 127.807,Z 532.289,A -85,B 0,C 180,E1 -25304.526,E2 -25304.526} C_VEL
LIN {X 0,Y 127.932,Z 529.727,A -85,B 0,C 180,E1 -25306.9,E2 -25306.9} C_VEL
LIN {X 0,Y 126.893,Z 525.015,A -85,B 0,C 180,E1 -25310.791,E2 -25310.791} C_VEL
LIN {X 0,Y 126.231,Z 519.715,A -85,B 0,C 180,E1 -25314.579,E2 -25314.579} C_VEL
LIN {X 0,Y 126.931,Z 516.144,A -85,B 0,C 180,E1 -25316.705,E2 -25316.705} C_VEL
LIN {X 0,Y 128.943,Z 510.786,A -85,B 0,C 180,E1 -25319.375,E2 -25319.375} C_VEL
LIN {X 0,Y 132.423,Z 501.843,A -85,B 0,C 180,E1 -25322.954,E2 -25322.954} C_VEL
LIN {X 0,Y 135.955,Z 492.008,A -85,B 0,C 180,E1 -25326.015,E2 -25326.015} C_VEL
LIN {X 0,Y 139.555,Z 481.244,A -85,B 0,C 180,E1 -25328.549,E2 -25328.549} C_VEL
LIN {X 0,Y 142.873,Z 469.133,A -85,B 0,C 180,E1 -25330.674,E2 -25330.674} C_VEL
LIN {X 0,Y 145.616,Z 456.486,A -85,B 0,C 180,E1 -25332.272,E2 -25332.272} C_VEL
LIN {X 0,Y 147.558,Z 444.057,A -85,B 0,C 180,E1 -25333.341,E2 -25333.341} C_VEL
LIN {X 0,Y 148.873,Z 427.799,A -85,B 0,C 180,E1 -25334.175,E2 -25334.175} C_VEL
LIN {X 0,Y 150.813,Z 397.525,A -85,B 0,C 180,E1 -25335.418,E2 -25335.418} C_VEL
LIN {X 0,Y 150.113,Z 386.943,A -85,B 0,C 180,E1 -25336.31,E2 -25336.31} C_VEL
LIN {X 0,Y 145.518,Z 373.854,A -85,B 0,C 180,E1 -25338.806,E2 -25338.806} C_VEL
LIN {X 0,Y 140.746,Z 363.066,A -85,B 0,C 180,E1 -25341.492,E2 -25341.492} C_VEL
LIN {X 0,Y 137.271,Z 357.116,A -85,B 0,C 180,E1 -25343.503,E2 -25343.503} C_VEL
LIN {X 0,Y 132.378,Z 349.876,A -85,B 0,C 180,E1 -25346.576,E2 -25346.576} C_VEL
LIN {X 0,Y 129.696,Z 346.024,A -85,B 0,C 180,E1 -25348.448,E2 -25348.448} C_VEL
LIN {X 0,Y 126.766,Z 342.523,A -85,B 0,C 180,E1 -25350.619,E2 -25350.619} C_VEL
LIN {X 0,Y 125.867,Z 340.78,A -85,B 0,C 180,E1 -25351.399,E2 -25351.399} C_VEL
LIN {X 0,Y 123.428,Z 338.811,A -85,B 0,C 180,E1 -25353.358,E2 -25353.358} C_VEL
LIN {X 0,Y 122.136,Z 336.148,A -85,B 0,C 180,E1 -25354.66,E2 -25354.66} C_VEL
LIN {X 0,Y 121.962,Z 335.291,A -85,B 0,C 180,E1 -25354.964,E2 -25354.964} C_VEL
LIN {X 0,Y 122.044,Z 335.284,A -85,B 0,C 180,E1 -25359.786,E2 -25359.786} C_VEL
LIN {X 0,Y 122.361,Z 335.212,A -85,B 0,C 180,E1 -25367.526,E2 -25367.526} C_VEL
LIN {X 0,Y 122.443,Z 335.201,A -85,B 0,C 180,E1 -25370.084,E2 -25370.084} C_VEL
LIN {X 0,Y 122.601,Z 335.191,A -85,B 0,C 180,E1 -25376.713,E2 -25376.713} C_VEL
LIN {X 0,Y 123.037,Z 335.123,A -85,B 0,C 180,E1 -25379.999,E2 -25379.999} C_VEL
LIN {X 0,Y 122.402,Z 335.222,A -85,B 0,C 180,E1 -25386.778,E2 -25386.778} C_VEL
LIN {X 0,Y 122.308,Z 335.227,A -85,B 0,C 180,E1 -25392.362,E2 -25392.362} C_VEL
LIN {X 0,Y 122.092,Z 335.268,A -85,B 0,C 180,E1 -25396.726,E2 -25396.726} C_VEL
LIN {X 0,Y 122.024,Z 335.265,A -85,B 0,C 180,E1 -25402.855,E2 -25402.855} C_VEL
LIN {X 0,Y 121.937,Z 335.279,A -85,B 0,C 180,E1 -25407.457,E2 -25407.457} C_VEL
LIN {X 0,Y 121.896,Z 335.27,A -85,B 0,C 180,E1 -25411.258,E2 -25411.258} C_VEL
LIN {X 0,Y 121.89,Z 335.296,A -85,B 0,C 180,E1 -25415.635,E2 -25415.635} C_VEL
LIN {X 0,Y 122.682,Z 337.798,A -85,B 0,C 180,E1 -25416.553,E2 -25416.553} C_VEL
LIN {X 0,Y 124.486,Z 339.986,A -85,B 0,C 180,E1 -25418.143,E2 -25418.143} C_VEL
LIN {X 0,Y 125.987,Z 341.092,A -85,B 0,C 180,E1 -25419.309,E2 -25419.309} C_VEL
LIN {X 0,Y 127.837,Z 344.173,A -85,B 0,C 180,E1 -25420.83,E2 -25420.83} C_VEL
LIN {X 0,Y 129.704,Z 346.181,A -85,B 0,C 180,E1 -25422.166,E2 -25422.166} C_VEL
LIN {X 0,Y 132.285,Z 349.844,A -85,B 0,C 180,E1 -25423.965,E2 -25423.965} C_VEL
LIN {X 0,Y 136.385,Z 355.799,A -85,B 0,C 180,E1 -25426.565,E2 -25426.565} C_VEL
LIN {X 0,Y 142.109,Z 364.766,A -85,B 0,C 180,E1 -25429.8,E2 -25429.8} C_VEL
LIN {X 0,Y 147.815,Z 375.61,A -85,B 0,C 180,E1 -25432.754,E2 -25432.754} C_VEL
LIN {X 0,Y 151.647,Z 383.938,A -85,B 0,C 180,E1 -25434.607,E2 -25434.607} C_VEL
LIN {X 0,Y 148.477,Z 431.576,A -85,B 0,C 180,E1 -25436.635,E2 -25436.635} C_VEL
LIN {X 0,Y 146.776,Z 445.495,A -85,B 0,C 180,E1 -25437.773,E2 -25437.773} C_VEL
LIN {X 0,Y 144.502,Z 457.89,A -85,B 0,C 180,E1 -25439.292,E2 -25439.292} C_VEL
LIN {X 0,Y 141.677,Z 468.867,A -85,B 0,C 180,E1 -25441.077,E2 -25441.077} C_VEL
LIN {X 0,Y 138.072,Z 480.349,A -85,B 0,C 180,E1 -25443.554,E2 -25443.554} C_VEL
LIN {X 0,Y 134.51,Z 490.663,A -85,B 0,C 180,E1 -25446.523,E2 -25446.523} C_VEL
LIN {X 0,Y 131.245,Z 499.103,A -85,B 0,C 180,E1 -25449.632,E2 -25449.632} C_VEL
LIN {X 0,Y 127.502,Z 508.24,A -85,B 0,C 180,E1 -25454.003,E2 -25454.003} C_VEL
LIN {X 0,Y 124.497,Z 515.594,A -85,B 0,C 180,E1 -25458.606,E2 -25458.606} C_VEL
LIN {X 0,Y 122.243,Z 521.493,A -85,B 0,C 180,E1 -25463.399,E2 -25463.399} C_VEL
LIN {X 0,Y 120.626,Z 526.16,A -85,B 0,C 180,E1 -25468.332,E2 -25468.332} C_VEL
LIN {X 0,Y 119.759,Z 530.08,A -85,B 0,C 180,E1 -25473.952,E2 -25473.952} C_VEL
LIN {X 0,Y 119.167,Z 532.947,A -85,B 0,C 180,E1 -25480.192,E2 -25480.192} C_VEL
LIN {X 0,Y 119.851,Z 534.537,A -85,B 0,C 180,E1 -25487.051,E2 -25487.051} C_VEL
LIN {X 0,Y 121.077,Z 534.652,A -85,B 0,C 180,E1 -25491.763,E2 -25491.763} C_VEL
LIN {X 0,Y 123.248,Z 533.823,A -85,B 0,C 180,E1 -25497.142,E2 -25497.142} C_VEL
LIN {X 0,Y 125.101,Z 532.782,A -85,B 0,C 180,E1 -25500.373,E2 -25500.373} C_VEL
LIN {X 0,Y 128.337,Z 530.532,A -85,B 0,C 180,E1 -25504.773,E2 -25504.773} C_VEL
LIN {X 0,Y 132.682,Z 526.942,A -85,B 0,C 180,E1 -25509.467,E2 -25509.467} C_VEL
LIN {X 0,Y 137.575,Z 522.372,A -85,B 0,C 180,E1 -25513.603,E2 -25513.603} C_VEL
LIN {X 0,Y 144.088,Z 515.375,A -85,B 0,C 180,E1 -25518.06,E2 -25518.06} C_VEL
LIN {X 0,Y 150.329,Z 507.753,A -85,B 0,C 180,E1 -25521.544,E2 -25521.544} C_VEL
LIN {X 0,Y 155.922,Z 499.918,A -85,B 0,C 180,E1 -25524.227,E2 -25524.227} C_VEL
LIN {X 0,Y 161.783,Z 490.279,A -85,B 0,C 180,E1 -25526.746,E2 -25526.746} C_VEL
LIN {X 0,Y 167.197,Z 479.501,A -85,B 0,C 180,E1 -25528.921,E2 -25528.921} C_VEL
LIN {X 0,Y 171.897,Z 468.401,A -85,B 0,C 180,E1 -25530.564,E2 -25530.564} C_VEL
LIN {X 0,Y 175.442,Z 457.667,A -85,B 0,C 180,E1 -25531.8,E2 -25531.8} C_VEL
LIN {X 0,Y 178.646,Z 444.732,A -85,B 0,C 180,E1 -25532.876,E2 -25532.876} C_VEL
LIN {X 0,Y 180.822,Z 432.005,A -85,B 0,C 180,E1 -25533.561,E2 -25533.561} C_VEL
